// TwinCAT 3 PLC project VFD
// Title: Modbus
// Company: HuynhPhuc
// ProjectVersion: 0.0.0.0
// ProgramVersion: 3.1.4024.0
// libraries:
//   Tc2_ModbusRTU, * (Beckhoff Automation GmbH)
//   Tc2_Standard, * (Beckhoff Automation GmbH)
//   Tc2_System, * (Beckhoff Automation GmbH)
//   Tc2_Utilities, * (Beckhoff Automation GmbH)
//   Tc3_Module, * (Beckhoff Automation GmbH)
// project tree:
//   / Class Diagram.TcCD (not stored), GVL.TcGVL, Machine.TcTTO
//   DUT/Common/ U_Word2Int.TcDUT (not stored)
//   DUT/File Logger/ E_FileLoggerAddLogsState.TcDUT, E_FileLoggerInitState.TcDUT (not stored), E_FileLoggerSetNewPathState.TcDUT (not stored), E_FileLoggerState.TcDUT (not stored)
//   DUT/M_Driver/ E_VfdMdriverFaultInfor.TcDUT (not stored)
//   DUT/Universal_Modbus/ E_ModbusFunction.TcDUT, E_ModBusMasterState.TcDUT, E_ModbusMasterStateRun.TcDUT
//   DUT/VFD/ E_VFD_State.TcDUT, E_VFD_Status.TcDUT (not stored)
//   DUT/Visu/ E_VisuCtrlVfdState.TcDUT (not stored), ST_VisuCtrlVfdFrame.TcDUT (not stored)
//   FC/ FC_ScaleValue.TcPOU (not stored), FUN_MergeLongStrings10.TcPOU, FUN_MergeStrings10.TcPOU, FUN_MergeStrings3.TcPOU, FUN_MergeStrings4.TcPOU, FUN_MergeStrings5.TcPOU, FUN_MergeStrings6.TcPOU, F_InRange.TcPOU
//   POUs/EmkoTemperature/ FB_TemperatureRelativeHumiditySensor_Emko.TcPOU
//   POUs/File Logger/ FB_FileLogger.TcPOU, I_FileLogger.TcIO (not stored)
//   POUs/ Prg_Machine.TcPOU
//   POUs/Universal Modbus RTU/ FB_ModbusMaster.TcPOU, FB_ModbusSlave.TcPOU, I_ModbusSlave.TcIO
//   POUs/VFD/ FB_UniversalVFDModbus.TcPOU, FB_VFD_ABB_ACS480.TcPOU, FB_VFD_Mdriver.TcPOU, I_UniversalVFD.TcIO
//   TEST/ FB_ModbusMaster_Test.TcPOU, FB_ModbusSlave_Test.TcPOU, FB_UniversalVFDModbus_Ex.TcPOU, FB_UniversalVFDModbus_Test.TcPOU, PGR_Test.TcPOU, README.TcPOU
// real-time tasks:
//   TASK Machine: cycle T#10ms, priority 20, ADS port 350
// I/O:
//   DEVICE Device 1 (NOV-DP-RAM) (disabled)
//   DEVICE Device 4 (COM Port) (disabled)

CONFIGURATION VFD
    RESOURCE PLC ON TwinCAT3
        TASK Machine(INTERVAL := T#10ms, PRIORITY := 20);
    END_RESOURCE
END_CONFIGURATION

// ---- DUT/File Logger/E_FileLoggerAddLogsState.TcDUT
{attribute 'strict'}
TYPE E_FileLoggerAddLogsState :
(
	FILE_LOGGER_ADD_LOGS_OPEN 			:= 0,	(* Opening file *)
	FILE_LOGGER_ADD_LOGS_WRITTE			:= 10,	(* Writting log from buffer to file *)
	FILE_LOGGER_ADD_LOGS_WRITTE_DONE	:= 20,	(* Writting log from buffer to file done *)
	FILE_LOGGER_ADD_LOGS_CLOSE 			:= 30,	(* Closing file *)
	FILE_LOGGER_ADD_LOGS_CLEAR			:= 40	(* Clearing buffer *)
);
END_TYPE

// ---- DUT/Universal_Modbus/E_ModbusFunction.TcDUT
{attribute 'qualified_only'}
TYPE E_ModbusFunction :
(	
	ReadCoils	:= 1,
	ReadDisCreteInputs := 2,
	ReadHoldingRegisters := 3, 
	ReadInputRegisters := 4,
	WriteSingleCoil := 5,
	WriteSingleRegister := 6,
	WriteMultipleCoils := 15,
	WriteMultipleRegisters := 16
) WORD;
END_TYPE

// ---- DUT/Universal_Modbus/E_ModBusMasterState.TcDUT
{attribute 'qualified_only'}
{attribute 'strict'}
TYPE E_ModBusMasterState :
(
	Uninitialized := 0,//0
	Initializing := 10,//10
	Ready	:= 20	,//20
	Running		:= 30,//30
	Stop		:= 200,//200
	Stop_done	:= 210//210
	
);
END_TYPE

// ---- DUT/Universal_Modbus/E_ModbusMasterStateRun.TcDUT
{attribute 'qualified_only'}
{attribute 'strict'}
TYPE E_ModbusMasterStateRun :
(
	CheckNumberSlaveRegistered 	:=0, 
	SetParametersRead 	:= 10,
	SendRequestRead		:= 20,
	WaitReadRespond	:= 40,
	ConvertRawData	:= 50,
	ReturnReadDone		:=60,
	
	SetParametersWrite 	:= 70,
	SendRequestWrite	:= 80,
	WaitWriteRespond := 90,
	ReturnWriteDone	:=120,

	
	notKnow			:= 210

);
END_TYPE

// ---- DUT/VFD/E_VFD_State.TcDUT
{attribute 'strict'}
{attribute 'to_string'}
TYPE E_VFD_State :
(
	VFD_ABORTING := -50,
	VFD_UNINITIALIZED := 0,
	VFD_INITIALIZING	:= 10,
	VFD_READY_INITIALIZED := 20,
	VFD_IDLE		:= 30,
	VFD_RUN_FORWARD	:= 40,
	VFD_RUN_FORWARD_DONE	:= 45,
	VFD_RUN_REVERSE	:= 50,
	VFD_RUN_REVERSE_DONE := 55,
	VFD_STOP		:= 60,
	VFD_STOP_DONE	:= 70,
	VFD_RESET	:= 80,
	VFD_RESET_DONE	:= 90
)INT;
END_TYPE

// ---- GVL.TcGVL

VAR_GLOBAL
	
	fbMachineLogger 						: FB_FileLogger;
	fbMachineTime							: FB_LocalSystemTime; 			
END_VAR

// ---- POUs/Universal Modbus RTU/I_ModbusSlave.TcIO
INTERFACE I_ModbusSlave

PROPERTY AddressRead : POINTER TO WORD
GET
END_GET
END_PROPERTY

PROPERTY AddressWrite : Pointer to Word
GET
END_GET
END_PROPERTY

METHOD Convert : BOOL
VAR_INPUT
	iRegionNo	:	INT;
	pReadData	:	POINTER TO word;
END_VAR
END_METHOD

METHOD FirstCycle 
VAR_INPUT
	sName : STRING;
	iUnitID : BYTE ; // modbus address of the device : 1- 255
END_VAR
END_METHOD

PROPERTY ModbusErrorID : MODBUS_ERRORS
GET
END_GET
SET
END_SET
END_PROPERTY

PROPERTY Name : STRING
GET
END_GET
SET
END_SET
END_PROPERTY

PROPERTY NumAddRegionRead : UINT
GET
END_GET
END_PROPERTY

PROPERTY NumAddRegionWrite : Uint
GET
END_GET
END_PROPERTY

PROPERTY UnitID : BYTE
GET
END_GET
SET
END_SET
END_PROPERTY

END_INTERFACE

// ---- POUs/VFD/I_UniversalVFD.TcIO
INTERFACE I_UniversalVFD


PROPERTY Active : REFERENCE TO  bool
GET
END_GET
END_PROPERTY

PROPERTY AcVoltageToMotor : Reference to lreal
GET
END_GET
END_PROPERTY


PROPERTY Busy : reference to bool
GET
END_GET
END_PROPERTY

PROPERTY Current : reference to lreal
GET
END_GET
END_PROPERTY

PROPERTY DcVoltage : Reference to lreal
GET
END_GET
END_PROPERTY


PROPERTY Error : REFERENCE to bool
GET
END_GET
END_PROPERTY


PROPERTY ErrorID : reference to UDINT
GET
END_GET
END_PROPERTY

PROPERTY HzActual : REFERENCE TO  LReal
GET
END_GET
END_PROPERTY

PROPERTY HzControl : reference to LReal
GET
END_GET
END_PROPERTY


PROPERTY InHz : bool
GET
END_GET
END_PROPERTY

PROPERTY isRunForward : bool
GET
END_GET
END_PROPERTY


PROPERTY IsRunning : bool
GET
END_GET
END_PROPERTY

PROPERTY isRunReverse : bool
GET
END_GET
END_PROPERTY

PROPERTY isStop : bool
GET
END_GET
END_PROPERTY

METHOD MR_Abort : BOOL
VAR_INPUT
END_VAR
END_METHOD

METHOD MR_Init : bool
VAR_INPUT
END_VAR
END_METHOD

METHOD MR_Reset : BOOL
VAR_INPUT
END_VAR
END_METHOD

//must stop before call run reverse or forward
METHOD MR_RunForward : BOOL// carefully about this state , it only into run forward if estatus = VFD_STATUS_RUNNING_FORWARD or it return True
VAR_INPUT
	hz : LREAL;
END_VAR
END_METHOD

METHOD MR_RunReverse : BOOL// must stop before call run reverse or forward
VAR_INPUT
	hz : LREAL; // >0 and < 50;
END_VAR
END_METHOD

METHOD MR_Stop : BOOL
VAR_INPUT
END_VAR
END_METHOD

PROPERTY Name : STRING
GET
END_GET
SET
END_SET
END_PROPERTY


PROPERTY Overload : reference TO BOOL
GET
END_GET
END_PROPERTY


PROPERTY PowerKw : REFERENCE TO LREAL
GET
END_GET
END_PROPERTY

PROPERTY Speed : Reference to lreal
GET
END_GET
END_PROPERTY


PROPERTY State : reference to E_Vfd_State
GET
END_GET
END_PROPERTY


PROPERTY Status : reference to E_VFD_Status
GET
END_GET
END_PROPERTY

PROPERTY timeStopDelay : time
GET
END_GET
SET
END_SET
END_PROPERTY

PROPERTY Torque : reference to lreal
GET
END_GET
END_PROPERTY

PROPERTY TotalKwh : reference to lreal
GET
END_GET
END_PROPERTY

PROPERTY Warning : reference to bool
GET
END_GET
END_PROPERTY

END_INTERFACE

// ---- POUs/File Logger/FB_FileLogger.TcPOU
(* 
:Description: This function block allows to log the data to txt file
*)
FUNCTION_BLOCK FB_FileLogger IMPLEMENTS I_FileLogger
VAR CONSTANT
	iBUFFER_SIZE : UINT := 255;
END_VAR
VAR
	sName : STRING;
	
	(* First cycle bits used for selecting file logging mode *)
	bAddTimeStamp				: BOOL;
	bAddHeader					: BOOL;
	
	(* Internal status *)
	bActive 					: BOOL;						(*  *)
	bBusy						: BOOL;						(*  *)
	bError						: BOOL;						(*  *)
	iErrorID					: UDINT;					(*  *)
	
	eFileLoggerState 			: E_FileLoggerState;		(*  *)
	eFileLoggerInitState 		: E_FileLoggerInitState;	(*  *)
	eFileLoggerAddLogsState		: E_FileLoggerAddLogsState; (*  *)
	eFileLoggerSetNewPathState 	: E_FileLoggerSetNewPathState;
	
	(* Internal parameters *)
	sFileName 					: STRING;					(*  *)
	sFileDir					: STRING;					(*  *)
	sFilePath					: STRING;					(*  *)
	
	hFile						: UINT;						(*  *)
	sAmsNetId					: T_AmsNetID;				(*  *)
	stTime						: TIMESTRUCT;				(*  *)
	sTime						: STRING;					(*  *)
	sFileDate					: STRING;									(*  *)
	sLogMessage					: STRING;									(*  *)
	
	(* Buffer arrays *)
	iCurrentBufferLine			: UINT := 1;								(*  *)
	iCurrentBufferLineForFile	: UINT := 1;								(*  *)
	arrMessageBuffer 			: ARRAY [1..iBUFFER_SIZE] OF STRING(300);	(*  *)
	arrMessageBufferPresence	: ARRAY [1..iBUFFER_SIZE] OF BOOL(255);		(*  *)
	
	(* Function blocks - time handling*)
	//fbGetTime					: NT_GetTime;				(*  *)
	
	(* Function blocks - file handling *)
	fbFileOpen					: FB_FileOpen;				(*  *)
	fbFileClose					: FB_FileClose;				(*  *)
	fbCreateDir					: FB_CreateDir;				(*  *)
	fbFilePuts					: FB_FilePuts;				(*  *)
END_VAR

bActive := eFileLoggerState >= FILE_LOGGER_READY;

IF fbMachineTime.bValid THEN
	stTime := fbMachineTime.systemTime;
	sTime := SYSTEMTIME_TO_STRING(stTime);
	
END_IF

StateMachine();

PROPERTY Active : REFERENCE TO BOOL
GET
Active REF= bActive;
END_GET
END_PROPERTY

PROPERTY AmsNetId : STRING
GET
AmsNetID := sAmsNetId;
END_GET
SET
sAmsNetId := AmsNetId;
END_SET
END_PROPERTY

PROPERTY Busy : REFERENCE TO BOOL
GET
Busy REF= bBusy;
END_GET
END_PROPERTY

PROPERTY Error : REFERENCE TO BOOL
GET
Error REF= bError;
END_GET
END_PROPERTY

PROPERTY ErrorID : REFERENCE TO UDINT
GET
ErrorID REF= iErrorID;
END_GET
END_PROPERTY

PROPERTY FileDir : STRING
GET
FileDir := sFileDir;
END_GET
SET
sFileDir := FileDir;
END_SET
END_PROPERTY

PROPERTY FileName : STRING
GET
FileName := sFileName;
END_GET
SET
sFileName := FileName;
END_SET
END_PROPERTY

METHOD M_ResetParameters : BOOL
VAR_INPUT
END_VAR
fbCreateDir( bExecute := FALSE);
fbFileOpen( bExecute := FALSE);
fbFilePuts( bExecute := FALSE);
fbFileClose( bExecute := FALSE);

FOR iCurrentBufferLine := 1 TO iBUFFER_SIZE BY 1 DO
	MEMSET(ADR(arrMessageBuffer[iCurrentBufferLine]),0,SIZEOF(arrMessageBuffer[iCurrentBufferLine]));
	arrMessageBufferPresence[iCurrentBufferLine] := FALSE;
END_FOR

iCurrentBufferLine := 1;
iCurrentBufferLineForFile := 1;

bError 		:= FALSE;
iErrorID 	:= 0;

MEMSET(ADR(sLogMessage),0,SIZEOF(sLogMessage));

eFileLoggerInitState := 0;
eFileLoggerAddLogsState := 0;
END_METHOD

METHOD M_SetNewPath : BOOL
VAR_INPUT
END_VAR
CASE eFileLoggerSetNewPathState OF
	FILE_LOGGER_SET_NEW_PATH_CHANGE_PATH:
		M_SetNewPath := FALSE;
		sFilePath := CONCAT(STR1 := sFileDir, STR2 := sFileName);
		
		eFileLoggerSetNewPathState := FILE_LOGGER_SET_NEW_PATH_DONE;
	
	FILE_LOGGER_SET_NEW_PATH_DONE:
		M_SetNewPath := TRUE;
		eFileLoggerSetNewPathState := FILE_LOGGER_SET_NEW_PATH_CHANGE_PATH;
			
END_CASE
END_METHOD

METHOD MR_Abort : BOOL
IF eFileLoggerState >= FILE_LOGGER_READY THEN
	bBusy := TRUE;
	MR_Abort := FALSE;
	eFileLoggerState := FILE_LOGGER_ABORTING;
	
ELSIF eFileLoggerState = FILE_LOGGER_UNINITIALIZED THEN
	bBusy := FALSE;
	MR_Abort := TRUE;
	
END_IF
END_METHOD

METHOD MR_AddLogs : BOOL
VAR_INPUT
	sLogMessage 	: STRING;		
	
END_VAR
VAR
	sCurrentTime 	: STRING;
	sCurrentDate	: STRING;
	sLog			: STRING(300);
	
END_VAR
IF iCurrentBufferLine >= iBUFFER_SIZE THEN	
	iCurrentBufferLine := 1;
		
ELSE
	sCurrentDate := LEFT(sTime,10);
	sCurrentTime := RIGHT(sTime,12);
	MEMSET(ADR(sLog),0,SIZEOF(sLog));
	
	IF bAddTimeStamp THEN
		sLog := FUN_MergeStrings6(sCurrentDate,'$t',sCurrentTime,'$t',sLogMessage,'$n'); 
	ELSE
		sLog := CONCAT(sLogMessage,'$n'); 
	END_IF
	
	MEMSET(ADR(arrMessageBuffer[iCurrentBufferLine]),0,SIZEOF(arrMessageBuffer[iCurrentBufferLine]));
	arrMessageBuffer[iCurrentBufferLine] := sLog;
	iCurrentBufferLine := iCurrentBufferLine + 1;
	
	MR_AddLogs := TRUE;
	
END_IF
END_METHOD

METHOD MR_FirstCycle : BOOL
VAR_INPUT
	sName 			: STRING;
	sFileDir		: STRING(255);
	sFileName		: STRING(255);
	sAmsNetId		: T_AmsNetID;
	bAddTimeStamp	: BOOL;
	bAddHeader		: BOOL;
END_VAR
THIS^.sName := sName;
THIS^.sFileDir := sFileDir;
THIS^.sFileName := sFileName;
THIS^.sAmsNetId := sAmsNetId;
THIS^.bAddTimeStamp := bAddTimeStamp;
THIS^.bAddHeader := bAddHeader;

M_SetNewPath();
END_METHOD

METHOD MR_Init : BOOL
VAR_INPUT
END_VAR
IF eFileLoggerState = FILE_LOGGER_UNINITIALIZED THEN
	bBusy := TRUE;
	MR_Init := FALSE;
	eFileLoggerState := FILE_LOGGER_INITIALIZING;
	
ELSIF eFileLoggerState >= FILE_LOGGER_READY THEN
	bBusy := FALSE;
	MR_Init := TRUE;
	
END_IF
END_METHOD

METHOD MR_Reset : BOOL
IF eFileLoggerState >= FILE_LOGGER_IDLE AND eFileLoggerState <> FILE_LOGGER_METHOD_DONE THEN
	bBusy := TRUE;
	MR_Reset := FALSE;
	eFileLoggerState := FILE_LOGGER_RESET;	

ELSIF eFileLoggerState = FILE_LOGGER_METHOD_DONE THEN
	bBusy := FALSE;
	MR_Reset := TRUE;

END_IF
END_METHOD

METHOD MR_SelectPath : BOOL
VAR_INPUT
	sFileDir								: STRING; 			(* CSV source file directory name *)
	sFileName 								: STRING; 			(* CSV source file name *)
END_VAR
IF eFileLoggerState = FILE_LOGGER_IDLE THEN
	THIS^.sFileDir := sFileDir;	
	THIS^.sFileName := sFileName;	
	bBusy := TRUE;
	MR_SelectPath := FALSE;
	eFileLoggerState := FILE_LOGGER_SELECT_PATH;
	
ELSIF eFileLoggerState = FILE_LOGGER_METHOD_DONE THEN
	bBusy := FALSE;
	MR_SelectPath := TRUE;
	
END_IF
END_METHOD

METHOD PROTECTED MS_Aborting
fbCreateDir( bExecute := FALSE);
fbFileOpen( bExecute := FALSE);
fbFilePuts( bExecute := FALSE);
fbFileClose( bExecute := FALSE);
//fbGetTime( START := FALSE);

FOR iCurrentBufferLine := 1 TO iBUFFER_SIZE BY 1 DO
	MEMSET(ADR(arrMessageBuffer[iCurrentBufferLine]),0,SIZEOF(arrMessageBuffer[iCurrentBufferLine]));
	arrMessageBufferPresence[iCurrentBufferLine] := FALSE;
	
END_FOR

iCurrentBufferLine := 1;
iCurrentBufferLineForFile := 1;

MEMSET(ADR(sTime),0,SIZEOF(sTime));
MEMSET(ADR(sFileDate),0,SIZEOF(sFileDate));
MEMSET(ADR(sLogMessage),0,SIZEOF(sLogMessage));

stTime.wDay 			:= 0;
stTime.wDayOfWeek 		:= 0;
stTime.wHour 			:= 0;
stTime.wMilliseconds 	:= 0;
stTime.wMinute 			:= 0;
stTime.wMonth 			:= 0;
stTime.wSecond 			:= 0;
stTime.wYear 			:= 0;

bActive		:= FALSE;
bBusy 		:= FALSE;
bError 		:= FALSE;
iErrorID 	:= 0;

eFileLoggerInitState := FILE_LOGGER_INIT_GET_TIME;
eFileLoggerAddLogsState := FILE_LOGGER_ADD_LOGS_OPEN;
eFileLoggerState := FILE_LOGGER_UNINITIALIZED;
END_METHOD

METHOD PROTECTED MS_AddLogs
CASE eFileLoggerAddLogsState OF
	FILE_LOGGER_ADD_LOGS_OPEN:
		IF NOT fbFileOpen.bError THEN
			fbFileOpen( sNetId 		:= sAmsNetId,
						sPathName 	:= FUN_MergeStrings4(sStr1 := sFilePath,'_',LEFT(sTime,10),'.txt'),
						bExecute 	:= TRUE,
						tTimeout	:= DEFAULT_ADS_TIMEOUT,
						nMode		:= FOPEN_MODEAPPEND OR FOPEN_MODEPLUS);
							
			IF NOT fbFileOpen.bBusy THEN
				fbFileOpen(bExecute := FALSE);				
				hFile := fbFileOpen.hFile;;
				eFileLoggerAddLogsState := FILE_LOGGER_ADD_LOGS_WRITTE;
			
			END_IF
		ELSE
			fbFileOpen( bExecute := FALSE);
			bError := fbFileOpen.bError;
			iErrorID := fbFileOpen.nErrId;

		END_IF
	

	FILE_LOGGER_ADD_LOGS_WRITTE:
		IF NOT fbFilePuts.bError THEN
			fbFilePuts( sNetId		:= sAmsNetId,
						hFile 		:= hFile,
						sLine 		:= arrMessageBuffer[iCurrentBufferLineForFile],
						bExecute 	:= TRUE,
						tTimeout 	:= DEFAULT_ADS_TIMEOUT);	
					
			IF NOT fbFilePuts.bBusy THEN				
				eFileLoggerAddLogsState := FILE_LOGGER_ADD_LOGS_WRITTE_DONE;
				
			END_IF
			
		ELSE
			fbFilePuts( bExecute := FALSE);
			bError := fbFilePuts.bError;
			iErrorID := fbFilePuts.nErrId;
			
		END_IF	

		
	FILE_LOGGER_ADD_LOGS_WRITTE_DONE:
		fbFilePuts( bExecute := FALSE);	
		iCurrentBufferLineForFile := iCurrentBufferLineForFile + 1;	
		
		IF iCurrentBufferLineForFile >= iBUFFER_SIZE THEN
			iCurrentBufferLineForFile := 1;
		ELSIF iCurrentBufferLineForFile < iCurrentBufferLine THEN
			eFileLoggerAddLogsState := FILE_LOGGER_ADD_LOGS_WRITTE;
		ELSIF iCurrentBufferLineForFile >= iCurrentBufferLine THEN
			eFileLoggerAddLogsState := FILE_LOGGER_ADD_LOGS_CLOSE;
		END_IF;

	
	FILE_LOGGER_ADD_LOGS_CLOSE:
		IF NOT fbFileClose.bError THEN
			fbFileClose(	sNetId := sAmsNetId,
							hFile := hFile,
							bExecute := TRUE,
							tTimeout := DEFAULT_ADS_TIMEOUT);
							
			IF NOT fbFileClose.bBusy THEN
				fbFileClose( bExecute := FALSE);
				eFileLoggerAddLogsState := FILE_LOGGER_ADD_LOGS_OPEN;
				eFileLoggerState := FILE_LOGGER_IDLE;

			END_IF
		ELSE
			bError := fbFileClose.bError;
			iErrorID := fbFileClose.nErrId;
			fbFileClose( bExecute := FALSE);
			
		END_IF
		
END_CASE
END_METHOD

METHOD PROTECTED MS_Idle
VAR_INPUT
END_VAR
IF iCurrentBufferLineForFile < iCurrentBufferLine THEN
	eFileLoggerState := FILE_LOGGER_ADD_LOGS;

END_IF
END_METHOD

METHOD PROTECTED MS_Initializing //C:\TwinCAT\log\filelog.txt
CASE eFileLoggerInitState OF
	FILE_LOGGER_INIT_CREATE_DIR:
		fbCreateDir(sNetId 		:= sAmsNetId,
					sPathName 	:= sFileDir,
					bExecute 	:= TRUE,
					tTimeout 	:= DEFAULT_ADS_TIMEOUT);
					
		IF NOT fbCreateDir.bBusy THEN
			eFileLoggerInitState := FILE_LOGGER_INIT_GET_TIME;
			fbCreateDir( bExecute := FALSE);
			
		END_IF
		
	FILE_LOGGER_INIT_GET_TIME:
		IF fbMachineTime.bValid THEN
			stTime := fbMachineTime.systemTime;
			sTime := SYSTEMTIME_TO_STRING(stTime);
			sFileDate := LEFT(sTime,10);
			eFileLoggerInitState := FILE_LOGGER_INIT_CREATE_FILE;
			
		END_IF
		
	FILE_LOGGER_INIT_CREATE_FILE:
		IF NOT fbFileOpen.bError THEN
			fbFileOpen( sNetId 		:= sAmsNetId,
						sPathName 	:= FUN_MergeStrings4(sFilePath,'_',LEFT(sTime,10),'.txt'),
						bExecute 	:= TRUE,
						tTimeout	:= DEFAULT_ADS_TIMEOUT,
						nMode		:= FOPEN_MODEAPPEND OR FOPEN_MODEPLUS);
							
			IF NOT fbFileOpen.bBusy THEN
				hFile := fbFileOpen.hFile;
				fbFileOpen(bExecute := FALSE);		
				
				IF bAddHeader THEN 
					eFileLoggerInitState := FILE_LOGGER_INIT_ADD_HEADER;
					
				ELSE
					eFileLoggerInitState := FILE_LOGGER_INIT_CLOSE_FILE;
					
				END_IF							
			END_IF
		ELSE
			bError := fbFileOpen.bError;
			iErrorID := fbFileOpen.nErrId;
			fbFileOpen( bExecute := FALSE);
			
		END_IF
		
	FILE_LOGGER_INIT_ADD_HEADER:
	
		IF NOT fbFilePuts.bError THEN
			fbFilePuts(	sNetId := sAmsNetId,
						hFile := hFile,
						sLine := CONCAT('----- Logger file initialized at ',CONCAT(LEFT(sTime,23),' ----- $n')),
						bExecute := TRUE,
						tTimeout := DEFAULT_ADS_TIMEOUT);

			IF NOT fbFilePuts.bBusy THEN
				eFileLoggerInitState := FILE_LOGGER_INIT_CLOSE_FILE;
				fbFilePuts( bExecute := FALSE);
				
			END_IF	
		ELSE
			bError := fbFilePuts.bError;
			iErrorID := fbFilePuts.nErrId;
			fbFilePuts( bExecute := FALSE);
			
		END_IF
	
	FILE_LOGGER_INIT_CLOSE_FILE:
		IF NOT fbFileClose.bError THEN
			fbFileClose( sNetId 		:= sAmsNetId,
							hFile 		:= hFile,
							bExecute 	:= TRUE,
							tTimeout 	:= DEFAULT_ADS_TIMEOUT);
							
			IF NOT fbFileClose.bBusy THEN
				eFileLoggerInitState := FILE_LOGGER_INIT_DONE;
				fbFileClose( bExecute := FALSE);
				
			END_IF
		ELSE
			bError := fbFileClose.bError;
			iErrorID := fbFileClose.nErrId;
			fbFileClose( bExecute := FALSE);
			
		END_IF
	
	FILE_LOGGER_INIT_DONE:
		eFileLoggerInitState := FILE_LOGGER_INIT_CREATE_DIR;
		eFileLoggerState := FILE_LOGGER_IDLE;
		
END_CASE
END_METHOD

METHOD PROTECTED MS_MethodDone
VAR_INPUT
END_VAR
IF NOT bBusy THEN
	eFileLoggerState := FILE_LOGGER_IDLE;

END_IF
END_METHOD

METHOD PROTECTED MS_Ready
VAR_INPUT
END_VAR
eFileLoggerState := FILE_LOGGER_IDLE;
END_METHOD

METHOD PROTECTED MS_Reset
VAR_INPUT
END_VAR
IF M_ResetParameters() THEN
	eFileLoggerState := FILE_LOGGER_METHOD_DONE;
	
END_IF
END_METHOD

METHOD MS_SelectPath : BOOL
VAR_INPUT
END_VAR
IF M_SetNewPath() THEN
	eFileLoggerState := FILE_LOGGER_METHOD_DONE;
	
END_IF
END_METHOD

METHOD PROTECTED MS_Uninitialized
;
END_METHOD

PROPERTY Name : STRING
GET
Name := sName;
END_GET
SET
sName := Name;
END_SET
END_PROPERTY

METHOD PROTECTED StateMachine
CASE eFileLoggerState OF
	FILE_LOGGER_UNINITIALIZED:
		MS_Uninitialized();
		
	FILE_LOGGER_INITIALIZING:
		MS_Initializing();
		
	FILE_LOGGER_IDLE:
		MS_Idle();
		
	FILE_LOGGER_ADD_LOGS:
		MS_AddLogs();	
		
	FILE_LOGGER_RESET:
		MS_Reset();
		
	FILE_LOGGER_METHOD_DONE:
		MS_MethodDone();
	
	FILE_LOGGER_ABORTING:
		MS_Aborting();
	
END_CASE
END_METHOD

END_FUNCTION_BLOCK

// ---- FC/FUN_MergeStrings6.TcPOU
(* 
:Description: This function is used to merge 6 strings
*)
FUNCTION FUN_MergeStrings6 : STRING(300)
VAR_INPUT
	sStr1	: STRING;		(* First string in merge row *)
	sStr2	: STRING;		(* Second string in merge row *)
	sStr3	: STRING;		(* Third string in merge row *)
	sStr4	: STRING;		(* Fourth string in merge row *)
	sStr5	: STRING;		(* Fifth string in merge row *)
	sStr6	: STRING;		(* Sixth string in merge row *)
END_VAR
(*
Version history:

+-------------+------------+----------------+----------+------------------------------------------+
|Date         | Version    | created under  | Author   | Remark                                   |
+=============+============+================+==========+==========================================+
|2022-06      | 1.0.0.0    | V3.1.4024.22   | ADS      | Function created    		              |
+-------------+------------+----------------+----------+------------------------------------------+

*)

FUN_MergeStrings6 := CONCAT(sStr1,sStr2);
FUN_MergeStrings6 := CONCAT(FUN_MergeStrings6, sStr3);
FUN_MergeStrings6 := CONCAT(FUN_MergeStrings6, sStr4);
FUN_MergeStrings6 := CONCAT(FUN_MergeStrings6, sStr5);
FUN_MergeStrings6 := CONCAT(FUN_MergeStrings6, sStr6);

END_FUNCTION

// ---- FC/FUN_MergeStrings4.TcPOU
(* 
:Description: This function is used to merge 5 strings
*)
FUNCTION FUN_MergeStrings4 : STRING
VAR_INPUT
	sStr1	: STRING;			(* Fifth string in merge row *)
	sStr2	: STRING;			(* Fourth string in merge row *)
	sStr3	: STRING;			(* Fourth string in merge row *)
	sStr4	: STRING;			(* Fourth string in merge row *)

END_VAR

FUN_MergeStrings4 := CONCAT(sStr1,sStr2);
FUN_MergeStrings4 := CONCAT(FUN_MergeStrings4,sStr3);
FUN_MergeStrings4 := CONCAT(FUN_MergeStrings4,sStr4);

END_FUNCTION

// ---- FC/FUN_MergeLongStrings10.TcPOU
(* 
:Description: This function is used to merge 10 long strings
*)
FUNCTION FUN_MergeLongStrings10 : STRING(2000)
VAR_INPUT
	sStr1	: STRING(2000);
	sStr2	: STRING(2000);
	sStr3	: STRING(2000);
	sStr4	: STRING(2000);
	sStr5	: STRING(2000);
	sStr6	: STRING(2000);
	sStr7	: STRING(2000);
	sStr8	: STRING(2000);
	sStr9	: STRING(2000);
	sStr10	: STRING(2000);
END_VAR
VAR
	sStrTemp1 :	STRING(2000);
	sStrTemp2 :	STRING(2000);
END_VAR
(*
Version history:

+-------------+------------+----------------+----------+------------------------------------------+
|Date         | Version    | created under  | Author   | Remark                                   |
+=============+============+================+==========+==========================================+
|2021-11      | 1.0.0.0    | V3.1.4024.22   | ADBO     | Function created		                  |
+-------------+------------+----------------+----------+------------------------------------------+

*)

CONCAT2(ADR(sStr1),ADR(sStr2),ADR(sStrTemp1),SIZEOF(sStrTemp1));
CONCAT2(ADR(sStrTemp1),ADR(sStr3),ADR(sStrTemp2),SIZEOF(sStrTemp2));
CONCAT2(ADR(sStrTemp2),ADR(sStr4),ADR(sStrTemp1),SIZEOF(sStrTemp1));
CONCAT2(ADR(sStrTemp1),ADR(sStr5),ADR(sStrTemp2),SIZEOF(sStrTemp2));
CONCAT2(ADR(sStrTemp2),ADR(sStr6),ADR(sStrTemp1),SIZEOF(sStrTemp1));
CONCAT2(ADR(sStrTemp1),ADR(sStr7),ADR(sStrTemp2),SIZEOF(sStrTemp2));
CONCAT2(ADR(sStrTemp2),ADR(sStr8),ADR(sStrTemp1),SIZEOF(sStrTemp1));
CONCAT2(ADR(sStrTemp1),ADR(sStr9),ADR(sStrTemp2),SIZEOF(sStrTemp2));
CONCAT2(ADR(sStrTemp2),ADR(sStr10),ADR(FUN_MergeLongStrings10),SIZEOF(FUN_MergeLongStrings10));

END_FUNCTION

// ---- FC/FUN_MergeStrings10.TcPOU
(* 
:Description: This function is used to merge 10 strings
*)
FUNCTION FUN_MergeStrings10 : STRING
VAR_INPUT
	sStr1	: STRING;		(* First string in merge row *)
	sStr2	: STRING;		(* Second string in merge row *)
	sStr3	: STRING;		(* Third string in merge row *)
	sStr4	: STRING(500);	(* Fourth string in merge row *)
	sStr5	: STRING(500);	(* Fifth string in merge row *)
	sStr6	: STRING(500);	(* Sixth string in merge row *)
	sStr7	: STRING(500);	(* Seventh string in merge row *)
	sStr8	: STRING;		(* Eight string in merge row *)
	sStr9	: STRING;		(* Ninth string in merge row *)
	sStr10	: STRING;		(* Tenth string in merge row *)
END_VAR
(*
Version history:

+-------------+------------+----------------+----------+------------------------------------------+
|Date         | Version    | created under  | Author   | Remark                                   |
+=============+============+================+==========+==========================================+
|2021-11      | 1.0.0.0    | V3.1.4024.22   | ADBO     | Function created      		              |
+-------------+------------+----------------+----------+------------------------------------------+

*)

FUN_MergeStrings10 := CONCAT(sStr1,sStr2);
FUN_MergeStrings10 := CONCAT(FUN_MergeStrings10,sStr3);
FUN_MergeStrings10 := CONCAT(FUN_MergeStrings10,sStr4);
FUN_MergeStrings10 := CONCAT(FUN_MergeStrings10,sStr5);
FUN_MergeStrings10 := CONCAT(FUN_MergeStrings10,sStr6);
FUN_MergeStrings10 := CONCAT(FUN_MergeStrings10,sStr7);
FUN_MergeStrings10 := CONCAT(FUN_MergeStrings10,sStr8);
FUN_MergeStrings10 := CONCAT(FUN_MergeStrings10,sStr9);
FUN_MergeStrings10 := CONCAT(FUN_MergeStrings10,sStr10);

END_FUNCTION

// ---- FC/FUN_MergeStrings3.TcPOU
(* 
:Description: This function is used to merge 5 strings
*)
FUNCTION FUN_MergeStrings3 : STRING
VAR_INPUT
	sStr1	: STRING;			(* Fifth string in merge row *)
	sStr2	: STRING;			(* Fourth string in merge row *)
	sStr3	: STRING;			(* Fourth string in merge row *)

END_VAR
(*
Version history:

+-------------+------------+----------------+----------+------------------------------------------+
|Date         | Version    | created under  | Author   | Remark                                   |
+=============+============+================+==========+==========================================+
|2022-06      | 1.0.0.0    | V3.1.4024.22   | ADS      | Function created    		              |
+-------------+------------+----------------+----------+------------------------------------------+

*)

FUN_MergeStrings3 := CONCAT(sStr1,sStr2);
FUN_MergeStrings3 := CONCAT(FUN_MergeStrings3,sStr3);

END_FUNCTION

// ---- FC/FUN_MergeStrings5.TcPOU
(* 
:Description: This function is used to merge 5 strings
*)
FUNCTION FUN_MergeStrings5 : STRING
VAR_INPUT
	sStr1	: STRING;		(* First string in merge row *)
	sStr2	: STRING;		(* Second string in merge row *)
	sStr3	: STRING;		(* Third string in merge row *)
	sStr4	: STRING;		(* Fourth string in merge row *)
	sStr5	: STRING;		(* Fifth string in merge row *)

END_VAR
(*
Version history:

+-------------+------------+----------------+----------+------------------------------------------+
|Date         | Version    | created under  | Author   | Remark                                   |
+=============+============+================+==========+==========================================+
|2021-11      | 1.0.0.0    | V3.1.4024.22   | ADBO     | Function created    		              |
+-------------+------------+----------------+----------+------------------------------------------+

*)

FUN_MergeStrings5 := CONCAT(sStr1,sStr2);
FUN_MergeStrings5 := CONCAT(FUN_MergeStrings5, sStr3);
FUN_MergeStrings5 := CONCAT(FUN_MergeStrings5, sStr4);
FUN_MergeStrings5 := CONCAT(FUN_MergeStrings5, sStr5);

END_FUNCTION

// ---- FC/F_InRange.TcPOU
FUNCTION F_InRange : BOOL // return true if value in [bound1, bound2] or in [bound2, bound1] else return false
VAR_INPUT
	bound1 : LREAL;
	bound2 : LREAL;
	value	: LREAL;
END_VAR
VAR
END_VAR

F_InRange := MIN(bound1, bound2)  <= value AND value <= MAX( bound1, bound2);

END_FUNCTION

// ---- POUs/EmkoTemperature/FB_TemperatureRelativeHumiditySensor_Emko.TcPOU
(*Odd or none parity bit only in model  PMDLx-x-0/0.1.1.x.x*)
FUNCTION_BLOCK FB_TemperatureRelativeHumiditySensor_Emko EXTENDS FB_ModbusSlave

VAR
	lrTemperature	: LREAL;
	lrRelativeHumidity : LREAL;
END_VAR

METHOD Convert : BOOL
VAR_INPUT
	iRegionNo	:	INT;
	pReadData	:	POINTER TO word;
END_VAR
CASE iRegionNo OF
	0:
		lrTemperature := WORD_TO_LREAL( pReadData[0])*0.01;
		lrRelativeHumidity := WORD_TO_LREAL( pReadData[1])*0.1;
END_CASE
END_METHOD

METHOD FirstCycle // must be call once time 
VAR_INPUT
	sName : STRING;
	iUnitID : BYTE ; // modbus address of the device : 1- 255
END_VAR
SUPER^.FirstCycle( sName := sName,
					iUnitID := iUnitID);
arrAddressRead[0][0] := 0;
arrAddressRead[0][1] := 2;
arrAddressRead[0][2] := E_ModbusFunction.ReadInputRegisters;
iNumAddRegionRead:= 1;
iNumAddRegionWrite := 0;
END_METHOD

PROPERTY RelativeHumidity : lreal
GET
RelativeHumidity := lrRelativeHumidity;
END_GET
END_PROPERTY

PROPERTY Temperature : lreal
GET
Temperature := lrTemperature;
END_GET
END_PROPERTY

END_FUNCTION_BLOCK

// ---- POUs/Universal Modbus RTU/FB_ModbusSlave.TcPOU
FUNCTION_BLOCK FB_ModbusSlave IMPLEMENTS I_ModbusSlave
VAR
	iUnitID	:	BYTE; // address of the Slave
	arrAddressRead	:	ARRAY [0..50] OF ARRAY [0..2] OF WORD;
	(*arrAddressRead[x][y]: +x : index of Region Read.  arrAddressRead[0]: the first region Read.
							+y:
								case y of
									0: Register address for Read
									1: Number of register for read
									2: Function Read
					 *)
	iNumAddRegionRead	:	UINT;
	
	arrAddressWrite		: ARRAY [0..20] OF ARRAY [0..10] OF WORD;// write Multiple or single register
	(* the 20 is max number of region write,
		arrAddressWrite[x][y] : +x: index of Region Read.  arrAddressRead[0]: the first region Read. 
								+y:
									case y of
										0 :  Register address for Write
										1 : number of register will be write => modbus master automatic choose Function Write( single Register or Multi Regiseter)
										2..9 : max 8 value for write
										10: Write Function : e.g E_ModbusFunction.WriteSingleCoil
															
	*)
	iNumAddRegionWrite	: UINT;
	
	bSwap			:		BOOL; // swap word receive from modbus master for convert
	sName			:		STRING;
	bFirstCycle 	: 		BOOL := TRUE;
	iModbusErrorID	:		MODBUS_ERRORS;
END_VAR

PROPERTY AddressRead : POINTER TO WORD
GET
AddressRead := ADR(arrAddressRead);
END_GET
END_PROPERTY

PROPERTY AddressWrite : POINTER TO WORD
GET
AddressWrite := ADR( arrAddressWrite);
END_GET
END_PROPERTY

METHOD Convert : BOOL
VAR_INPUT
	iRegionNo	:	INT;
	pReadData	:	POINTER TO word;
END_VAR
END_METHOD

METHOD FirstCycle // must be call once time 
VAR_INPUT
	sName : STRING;
	iUnitID : BYTE ; // modbus address of the device : 1- 255
END_VAR
THIS^.sName := sName;
THIS^.iUnitID := iUnitID;
END_METHOD

{attribute 'monitoring' := 'variable'}
PROPERTY ModbusErrorID : MODBUS_ERRORS
GET
ModbusErrorID := iModbusErrorID;
END_GET
SET
iModbusErrorID := ModbusErrorID;
END_SET
END_PROPERTY

PROPERTY Name : STRING
GET
Name := sName;
END_GET
SET
sName := Name;
END_SET
END_PROPERTY

PROPERTY NumAddRegionRead : UINT
GET
NumAddRegionRead := iNumAddRegionRead;
END_GET
END_PROPERTY

PROPERTY NumAddRegionWrite : UINT
GET
NumAddRegionWrite := iNumAddRegionWrite;
END_GET
END_PROPERTY

PROPERTY UnitID : BYTE
GET
UnitID := iUnitID;
END_GET
SET
iUnitID := UnitID;
END_SET
END_PROPERTY

END_FUNCTION_BLOCK

// ---- POUs/Prg_Machine.TcPOU
PROGRAM Prg_Machine
VAR
	fbModbusMaster	: FB_ModbusMaster;
	ABBAcs480 : FB_VFD_ABB_ACS480;
	Mdriver : fB_VFD_Mdriver;
	arrIfVFD : ARRAY[0..numberOfVFD-1] OF I_UniversalVFD;
	emkoSs	: FB_TemperatureRelativeHumiditySensor_Emko;
	bInit	: BOOL;
	bAbort : BOOL;
	bFirstCycle	: BOOL := TRUE;
	bModbusRun	: BOOL;
	hzControl	: LREAL;
	arrVfdState	: ARRAY [0..iVFDS_PER_PAGE-1] OF E_VisuCtrlVfdState; 
	arrVfdFrame	: ARRAY [0..iVFDS_PER_PAGE-1] OF ST_VisuCtrlVfdFrame;
	iloop		: UINT;
	lrTemp	: LREAL;
	lrhumidity	: LREAL;
END_VAR
VAR CONSTANT
	iVFDS_PER_PAGE : UINT := 2;
	numberOfVFD	: UINT := 2;
END_VAR

IF bFirstCycle THEN
	Mdriver.FirstCycle( sName := 'M_driver',
						iUnitID := 4 );
	ABBAcs480.FirstCycle( sName := 'ABB acs480',
							iUnitID := 5);			
	emkoSs.FirstCycle( sName := 'ss 01',
						iUnitID := 10);
	arrIfVFD[0] := Mdriver;
	arrIfVFD[1] := ABBAcs480;				
	IF fbModbusMaster.Init() THEN
		fbModbusMaster.RegisterSlave( ModbusSlave := ABBAcs480);
		fbModbusMaster.RegisterSlave( ModbusSlave := Mdriver);
		fbModbusMaster.RegisterSlave( ModbusSlave := emkoSs);
		fbModbusMaster.Timeout := 1000;
		bFirstCycle := FALSE;
	END_IF
END_IF
fbModbusMaster.Run();
fbModbusMaster();
Mdriver();
ABBAcs480();
lrTemp := emkoSs.Temperature;
lrhumidity := emkoSs.RelativeHumidity;
(*visu*)
FOR iloop := 0 TO numberOfVFD-1 DO
	arrVfdFrame[iLoop].lrCurrent		:= arrIfVFD[iloop].Current;
	arrVfdFrame[iLoop].bError			:= arrIfVFD[iloop].error;
	arrVfdFrame[iLoop].lrHz_actual		:= arrIfVFD[iloop].HzActual;
	arrVfdFrame[iLoop].eStatus			:= arrIfVFD[iloop].Status;
	arrVfdFrame[iLoop].sStatus			:= TO_STRING(arrVfdFrame[iLoop].eStatus);
	arrVfdFrame[iLoop].eState			:= arrIfVFD[iloop].State;
	arrVfdFrame[iloop].sState			:= TO_STRING(arrVfdFrame[iLoop].eState);
	arrVfdFrame[iloop].errorID			:= arrIfVFD[iloop].errorID;	
	arrVfdFrame[iloop].sName			:= arrIfVFD[iloop].Name;	
	IF arrVfdFrame[iLoop].btnReset THEN
		arrVfdFrame[iLoop].btnReset := FALSE;
		arrVfdState[iLoop] := VISU_CTRL_VFDS_RESET;
	END_IF
	
	IF arrVfdFrame[iLoop].btnAbort THEN
		arrVfdFrame[iLoop].btnAbort	:= FALSE;
		arrVfdState[iLoop] := VISU_CTRL_VFDS_ABORT;						
	END_IF	
	CASE arrVfdState[iLoop] OF
		
		VISU_CTRL_VFDS_WAIT_FOR_CMD:
			IF arrVfdFrame[iLoop].btnInit THEN
				arrVfdFrame[iLoop].btnInit	:= FALSE;
				arrVfdState[iLoop] := VISU_CTRL_VFDS_INIT;
				
			ELSIF arrVfdFrame[iLoop].btnStop THEN
				arrVfdFrame[iLoop].btnStop	:= FALSE;
				arrVfdState[iLoop] := VISU_CTRL_VFDS_STOP;
				
			ELSIF arrVfdFrame[iLoop].btnRunForward THEN
				arrVfdFrame[iLoop].btnRunForward	:= FALSE;
				arrVfdState[iLoop] := VISU_CTRL_VFDS_RUN_FORWARD;
				
			ELSIF arrVfdFrame[iLoop].btnRunReverse THEN
				arrVfdFrame[iLoop].btnRunReverse	:= FALSE;
				arrVfdState[iLoop] := VISU_CTRL_VFDS_RUN_REVERSE;						
				
			END_IF
			
		VISU_CTRL_VFDS_INIT:					
			arrIfVFD[iloop].MR_Init();
			IF arrIfVFD[iloop].Active AND NOT arrIfVFD[iloop].Busy THEN
				arrVfdState[iLoop] := VISU_CTRL_VFDS_WAIT_FOR_CMD;
			END_IF
			
		VISU_CTRL_VFDS_RESET:		 			
			arrIfVFD[iloop].MR_Reset();
			IF NOT arrIfVFD[iloop].Error AND NOT arrIfVFD[iloop].Busy THEN
				arrVfdState[iLoop] := VISU_CTRL_VFDS_WAIT_FOR_CMD;
			END_IF
		
		VISU_CTRL_VFDS_RUN_FORWARD:	
			arrIfVFD[iloop].MR_RunForward(arrVfdFrame[iLoop].lrHz_Control);		
			IF arrIfVFD[iloop].isRunForward AND NOT arrIfVFD[iloop].Busy THEN
				arrVfdState[iLoop] := VISU_CTRL_VFDS_WAIT_FOR_CMD;
			END_IF
		
		VISU_CTRL_VFDS_RUN_REVERSE:
			arrIfVFD[iloop].MR_RunReverse(arrVfdFrame[iLoop].lrHz_Control);
			IF arrIfVFD[iloop].isRunReverse AND NOT arrIfVFD[iloop].Busy THEN
				arrVfdState[iLoop] := VISU_CTRL_VFDS_WAIT_FOR_CMD;
			END_IF
			
		VISU_CTRL_VFDS_STOP:
			arrIfVFD[iloop].MR_Stop();
			IF arrIfVFD[iloop].isStop AND NOT arrIfVFD[iloop].Busy THEN
				arrVfdState[iLoop] := VISU_CTRL_VFDS_WAIT_FOR_CMD;
			END_IF
			
		VISU_CTRL_VFDS_ABORT:
			arrIfVFD[iloop].MR_Abort();
			IF NOT arrIfVFD[iloop].Active AND NOT arrIfVFD[iloop].Busy	THEN
				arrVfdState[iLoop] := VISU_CTRL_VFDS_WAIT_FOR_CMD;
			END_IF
					
	END_CASE
END_FOR

END_PROGRAM

// ---- POUs/Universal Modbus RTU/FB_ModbusMaster.TcPOU
FUNCTION_BLOCK FB_ModbusMaster //IMPLEMENTS I_UniversalUnit
VAR
	sName			:		STRING;
	bInitialized	:		BOOL;
	iScantime		:		UINT;
	iTimeout		:		UINT := 1000;//1000ms
	iErrorID		:		MODBUS_ERRORS;
	bBusy			: 		BOOL;
	bError			:		BOOL;
	iStepGeneral	: 		E_ModBusMasterState;
	iStepRunning	:		E_ModbusMasterStateRun;
	bFirstCycle		:		BOOL;
	bRun			:		BOOL;
	bStop			: 		BOOL;

	fbModbusMaster	: 		ModbusRtuMaster_PcCOM;
	//fbModbusMaster : 		ModbusRtuMasterV2_KL6x22B;
	ipModbusSlave	:		ARRAY [1..247] OF I_ModbusSlave;
	iAmountSlave	: 		UINT;
	
	iLoopSlave		:		UINT	:= 1;
	iLoopAdr		:		UINT;
	iQuantity 		: 		POINTER TO WORD;
	iMBAddr 		: 		POINTER TO WORD;
    arrData			: 		ARRAY [0..255] OF WORD;
	
	UnitId	: BYTE;
	Quantity	: WORD;
	MBAddr	: WORD;
	cbLength : UINT;
	pMemoryAddr	: POINTER TO BYTE;
	pDataWrite	: POINTER TO WORD;

	bexecute	: BOOL;
	
	tCalculateTimeRW	: TON;
	nNumberFaultRW	: UINT;
	eModbusFunction: E_ModbusFunction;
	peModbusFunction : POINTER TO WORD;
END_VAR

StateMachine();
bRun :=  iStepGeneral = E_ModBusMasterState.Running ;
bStop := iStepGeneral = E_ModBusMasterState.stop_done;
bInitialized := iStepGeneral >= E_ModBusMasterState.Ready;
iErrorID := fbModbusMaster.ErrorId;
tCalculateTimeRW(PT	:= T#10S); // for test how much time read write total

METHOD Abort : BOOL
bError := FALSE;
iErrorID := 0;
bError := FALSE;
iStepGeneral	:= E_ModBusMasterState.Uninitialized;
iStepRunning	:= E_ModbusMasterStateRun.CheckNumberSlaveRegistered;

iLoopSlave		:= 1;
iLoopAdr		:= 0;

fbModbusMaster(Execute := FALSE);

Abort := TRUE;
END_METHOD

PROPERTY AnyError : BOOL
GET
AnyError 	:= bError;
END_GET
END_PROPERTY

PROPERTY Busy : BOOL
GET
Busy := bBusy;
END_GET
END_PROPERTY

PROPERTY ErrorID : MODBUS_ERRORS
GET
ErrorID := iErrorID;
END_GET
END_PROPERTY

METHOD Init : BOOL
IF iStepGeneral = E_ModBusMasterState.Uninitialized THEN
	iStepGeneral := E_ModBusMasterState.Initializing;
END_IF

//Method output
	Init := (iStepGeneral >= E_ModBusMasterState.Ready);
END_METHOD

PROPERTY Initialized : BOOL
GET
Initialized := bInitialized;
END_GET
END_PROPERTY

PROPERTY Name : STRING
GET
Name := sName;
END_GET
SET
sName := Name;
END_SET
END_PROPERTY

PROPERTY ReadData : ARRAY [0..255] OF Word
GET
ReadData := arrData;
END_GET
END_PROPERTY

PROPERTY ReadDataSize : uint
GET
ReadDataSize := INT_TO_UINT(SIZEOF(arrData));
END_GET
END_PROPERTY

METHOD RegisterSlave : BOOL
VAR_INPUT
	ModbusSlave		:		I_ModbusSlave;
END_VAR
VAR
	iLoop	:	UINT;
	bExists	:	BOOL;
END_VAR
FOR iLoop := 1 TO iAmountSlave DO
	IF ipModbusSlave[iLoop] = ModbusSlave THEN
		bExists := TRUE;
		iLoop := iAmountSlave;// end loop for command
	END_IF
END_FOR 
IF NOT bExists THEN
	iAmountSlave := iAmountSlave + 1;
	ipModbusSlave[iAmountSlave] := ModbusSlave;
END_IF
END_METHOD

METHOD Reset : BOOL
bError := FALSE;
iErrorID := 0;
bError := FALSE;
iStepGeneral	:= E_ModBusMasterState.Uninitialized;
iStepRunning	:= E_ModbusMasterStateRun.CheckNumberSlaveRegistered;

iLoopSlave		:= 1;
iLoopAdr		:= 0;

fbModbusMaster.Execute := FALSE;

Reset := TRUE;
END_METHOD

METHOD Run : BOOL /// call from FB_modbus
IF (iStepGeneral = E_ModBusMasterState.Ready) THEN
	iStepGeneral := E_ModBusMasterState.Running;
END_IF

bRun := TRUE;
Run := (iStepGeneral >= E_ModBusMasterState.Running) AND (iStepGeneral < E_ModBusMasterState.stop);
END_METHOD

PROPERTY ScanTime : UINT
GET
ScanTime := iScantime;
END_GET
SET
iScantime := ScanTime;
END_SET
END_PROPERTY

METHOD protected StateInit : BOOL (*Unit is performing initialization*)
IF NOT bError THEN
	iStepGeneral := E_ModBusMasterState.Ready;
END_IF
END_METHOD

METHOD protected StateMachine : BOOL (*State machine of unit*)
CASE iStepGeneral OF
		E_ModBusMasterState.Uninitialized:  
			StateUninitialized();
	
		E_ModBusMasterState.Initializing: 
			StateInit();
	
		E_ModBusMasterState.Ready: 
			StateReady();
		
		E_ModBusMasterState.Running: 
			StateRunning();
						
		E_ModBusMasterState.stop:
			StateStopping();
			
		E_ModBusMasterState.stop_done:
			StateStoppingDone();
END_CASE
END_METHOD

METHOD protected StateReady : BOOL (* Unit is initialized*)
END_METHOD

METHOD PROTECTED StateRunning : BOOL (* Unit is uninitialized*)
VAR 
	

	
END_VAR
CASE iStepRunning OF
	E_ModbusMasterStateRun.CheckNumberSlaveRegistered: // Trigger
		IF iAmountSlave > 0 THEN
			iStepRunning := E_ModbusMasterStateRun.SetParametersRead;
		END_IF
					
	E_ModbusMasterStateRun.SetParametersRead: // Set parameters
		IF ipModbusSlave[iLoopSlave].NumAddRegionRead <> 0 
		AND iLoopAdr <= (ipModbusSlave[iLoopSlave].NumAddRegionRead - 1) 
		THEN
			iQuantity := ipModbusSlave[iLoopSlave].AddressRead + ((iLoopAdr * 3 + 1) * SIZEOF(WORD));// arrAddressRead[iloopAdr][1] in Slave
			iMBAddr := ipModbusSlave[iLoopSlave].AddressRead + ((iLoopAdr * 3) * SIZEOF(WORD));// arrAddressRead[iloopAdr][0] in Slave
			UnitID := ipModbusSlave[iLoopSlave].UnitID;
			Quantity :=	iQuantity^;
			MBAddr := iMBAddr^;
			cbLength := SIZEOF(arrData);
			pMemoryAddr	:= ADR(arrData);
			peModbusFunction := ipModbusSlave[iLoopSlave].AddressRead + ((iLoopAdr * 3 + 2) * SIZEOF(WORD)); // arrAddressRead[iloopAdr][2] in Slave
			eModbusFunction := peModbusFunction^;
			iStepRunning := E_ModbusMasterStateRun.SendRequestRead;
		ELSE 
			iLoopAdr := 0;
			iStepRunning := E_ModbusMasterStateRun.ReturnReadDone;
		END_IF

			
	E_ModbusMasterStateRun.SendRequestRead: // Send request
		CASE eModbusFunction OF
			E_ModbusFunction.ReadHoldingRegisters:
				fbModbusMaster.ReadRegs(
					UnitID:= UnitID, 
					Quantity:= Quantity, 
					MBAddr:= MBAddr, 
					cbLength:= cbLength, 
					pMemoryAddr:= pMemoryAddr, 
					Execute:= TRUE,
					Timeout:= UINT_TO_TIME(iTimeout),
					BUSY=> bBusy, 
					Error=> bError , 
					ErrorId=>iErrorId 
				);
			
			E_ModbusFunction.ReadInputRegisters:
				fbModbusMaster.ReadInputRegs(
					UnitID:= UnitID, 
					Quantity:= Quantity, 
					MBAddr:= MBAddr, 
					cbLength:= cbLength, 
					pMemoryAddr:= pMemoryAddr, 
					Execute:= TRUE,
					Timeout:= UINT_TO_TIME(iTimeout),
					BUSY=> bBusy, 
					Error=> bError , 
					ErrorId=>iErrorId 
				);
			
		END_CASE
		iStepRunning := E_ModbusMasterStateRun.WaitReadRespond;
						
	E_ModbusMasterStateRun.WaitReadRespond:
		fbModbusMaster.ReadRegs(Execute := FALSE);
		fbModbusMaster.ReadInputRegs(Execute := FALSE);
		ipModbusSlave[iLoopSlave].ModbusErrorID := iErrorID;
		IF NOT fbModbusMaster.BUSY AND NOT fbModbusMaster.Error THEN
			iStepRunning := E_ModbusMasterStateRun.ConvertRawData;
			nNumberFaultRW := 0;
		END_IF
		
		IF fbModbusMaster.Error AND NOT fbModbusMaster.BUSY THEN
			iStepRunning := E_ModbusMasterStateRun.ReturnReadDone;
		END_IF
	
	E_ModbusMasterStateRun.ConvertRawData: 
		ipModbusSlave[iLoopSlave].Convert(
			iRegionNo := iLoopAdr,
		 	pReadData := ADR(arrData)
		);
		iLoopAdr := iLoopAdr + 1;
		iStepRunning := E_ModbusMasterStateRun.CheckNumberSlaveRegistered;

	E_ModbusMasterStateRun.ReturnReadDone: // Return, done
		iStepRunning := E_ModbusMasterStateRun.SetParametersWrite;
		iLoopAdr := 0;

	E_ModbusMasterStateRun.SetParametersWrite :
		IF  ipModbusSlave[iLoopSlave].NumAddRegionWrite <> 0
		AND iLoopAdr <= ipModbusSlave[iLoopSlave].NumAddRegionWrite - 1 
		THEN // iLoopAdr start from 1
			iMBAddr := ipModbusSlave[iLoopSlave].AddressWrite + (iLoopAdr * 11 * SIZEOF(WORD));// return address word contain value address( modbus) 
			pDataWrite := ipModbusSlave[iLoopSlave].AddressWrite + ((iLoopAdr * 11 + 2) * SIZEOF(WORD));
			iQuantity := ipModbusSlave[iLoopSlave].AddressWrite + ((iLoopAdr * 11 + 1) * SIZEOF(WORD));
			peModbusFunction := ipModbusSlave[iLoopSlave].AddressWrite + ((iLoopAdr * 11 + 10) * SIZEOF(WORD));
			eModbusFunction := peModbusFunction^;
			UnitID 	:=		ipModbusSlave[iLoopSlave].UnitID;
			Quantity	:=	iQuantity^;
			MBAddr	:=		iMBAddr^;
			cbLength	:= 	Quantity * 2;
			pMemoryAddr	:= 	pDataWrite;
			iStepRunning := E_ModbusMasterStateRun.SendRequestWrite;
		ELSE 
			iStepRunning := E_ModbusMasterStateRun.ReturnWriteDone;
		END_IF

	E_ModbusMasterStateRun.SendRequestWrite :
		CASE eModbusFunction OF
			E_ModbusFunction.WriteMultipleCoils:
				fbModbusMaster.WriteMultipleCoils(
					UnitID:= UnitID, 
					Quantity:= Quantity, 
					MBAddr:= MBAddr, 
					cbLength:= cbLength, 
					pMemoryAddr:= pMemoryAddr, 
					Execute:=  true,
					Timeout:= 	UINT_TO_TIME(iTimeout),	
					BUSY=> bBusy, 
					Error=> bError , 
					ErrorId=>iErrorId 
				);
													
			E_ModbusFunction.WriteMultipleRegisters:
				fbModbusMaster.WriteRegs(
					UnitID:= UnitID, 
					Quantity:= Quantity, 
					MBAddr:= MBAddr, 
					cbLength:= cbLength, 
					pMemoryAddr:= pMemoryAddr, 
					Execute:= TRUE,
					Timeout:= UINT_TO_TIME(iTimeout),	
					BUSY=> bBusy, 
					Error=> bError , 
					ErrorId=>iErrorId 
				);
											
			E_ModbusFunction.WriteSingleCoil:
				fbModbusMaster.WriteSingleCoil(
					UnitID:= UnitID, 
					Quantity:= Quantity, 
					MBAddr:= MBAddr, 
					cbLength:= cbLength, 
					pMemoryAddr:= pMemoryAddr, 
					Execute:=  true,
					Timeout:= UINT_TO_TIME(iTimeout),	
					BUSY=> bBusy, 
					Error=> bError , 
					ErrorId=>iErrorId 
				);
			E_ModbusFunction.WriteSingleRegister:
				fbModbusMaster.WriteSingleRegister(
					UnitID:= UnitID, 
					Quantity:= Quantity, 
					MBAddr:= MBAddr, 
					cbLength:= cbLength, 
					pMemoryAddr:= pMemoryAddr, 
					Execute:=  true,
					Timeout:= 	UINT_TO_TIME(iTimeout),	
					BUSY=> bBusy, 
					Error=> bError , 
					ErrorId=>iErrorId 
				);
		END_CASE
		
		iStepRunning := E_ModbusMasterStateRun.WaitWriteRespond;
	
	E_ModbusMasterStateRun.WaitWriteRespond :
		fbModbusMaster.WriteMultipleCoils( Execute := FALSE);
		fbModbusMaster.WriteRegs( Execute := FALSE);
		fbModbusMaster.WriteSingleCoil( Execute := FALSE);	
		fbModbusMaster.WriteSingleRegister( Execute := FALSE);
		ipModbusSlave[iLoopSlave].ModbusErrorID := iErrorID;
		IF NOT fbModbusMaster.BUSY AND NOT fbModbusMaster.Error THEN
			iStepRunning := E_ModbusMasterStateRun.SetParametersWrite;
			nNumberFaultRW := 0;
			iLoopAdr := iLoopAdr + 1;
		END_IF
		IF fbModbusMaster.Error AND NOT fbModbusMaster.BUSY THEN
			iStepRunning := E_ModbusMasterStateRun.ReturnWriteDone ;
		END_IF
	
	 E_ModbusMasterStateRun.ReturnWriteDone :
		iLoopAdr := 0;
		iLoopSlave := iLoopSlave + 1;// next slave
		IF iLoopSlave > iAmountSlave THEN
			iLoopSlave := 1;
		END_IF
		THIS^.tCalculateTimeRW(in := FALSE);
		tCalculateTimeRW(in := TRUE);
		iStepRunning := E_ModbusMasterStateRun.CheckNumberSlaveRegistered;
		
END_CASE
END_METHOD

METHOD protected StateStopping : BOOL (* Unit is uninitialized*)
iStepGeneral	:= E_ModBusMasterState.Uninitialized;
iStepRunning	:= E_ModbusMasterStateRun.notKnow;

iLoopSlave		:= 1;
iLoopAdr		:= 0;

fbModbusMaster(Execute := FALSE);
END_METHOD

METHOD protected StateStoppingDone : BOOL (* Unit is uninitialized*)
IF NOT bStop THEN
	iStepGeneral := E_ModBusMasterState.Ready;
END_IF
END_METHOD

METHOD protected StateUninitialized : BOOL (* Unit is uninitialized*)
END_METHOD

METHOD protected Stop : BOOL
IF iStepGeneral >= E_ModBusMasterState.Running AND iStepGeneral < E_ModBusMasterState.stop THEN
	iStepGeneral := E_ModBusMasterState.stop;
END_IF
bStop := TRUE;

Stop := (iStepGeneral = E_ModBusMasterState.stop_done);
END_METHOD

PROPERTY Timeout : UINT // in milisecond, if not respond in this time , error will raise
GET
Timeout := iTimeout;
END_GET
SET
iTimeout := Timeout;
END_SET
END_PROPERTY

END_FUNCTION_BLOCK

// ---- POUs/VFD/FB_VFD_ABB_ACS480.TcPOU
FUNCTION_BLOCK FB_VFD_ABB_ACS480 EXTENDS FB_UniversalVFDModbus

VAR
	VFD_CTRL_RUN_EMERGENCY_STOP : WORD;
	TempData0: U_Word2Int;
END_VAR

SUPER^();

METHOD Convert : BOOL
VAR_INPUT
	iRegionNo	:	INT;
	pReadData	:	POINTER TO word;
END_VAR
CASE	iRegionNo OF

	0: // status
		IF pReadData[0].15 = TRUE THEN
			eVfdStatus := VFD_STATUS_FAULT;
			
		ELSIF (eVfdState = VFD_INITIALIZING
			OR eVfdState = VFD_READY_INITIALIZED)
			AND pReadData[0].0 = TRUE
			AND pReadData[0].1 = TRUE	
			AND pReadData[0].2 = TRUE
			THEN
			eVfdStatus :=  VFD_STATUS_READY_TO_RUN;
				
		ELSIF pReadData[0].3 = FALSE THEN
			eVfdStatus :=  VFD_STATUS_STOP;
			
		ELSIF pReadData[0].3 = TRUE	//run
			AND pReadData[0].10 = FALSE	// Drive reference is in the forward direction	
			AND pReadData[0].11 = FALSE//Drive is running in the forward direction
			THEN		
			eVfdStatus := VFD_STATUS_RUNNING_FORWARD;
		
		ELSIF pReadData[0].3 = TRUE	//run
			AND pReadData[0].10 = TRUE	// Drive reference is in the forward direction	
			AND pReadData[0].11 = TRUE//Drive is running in the forward direction
			THEN		
			eVfdStatus := VFD_STATUS_RUNNING_REVERSE;
		
		END_IF
	1: 
		TempData0.iWord := pReadData[0];
		lrHzActual		:= ABS(INT_TO_LREAL( TempData0.iInt)*0.0025);//50/20000;	
		lrCurrent		:= WORD_TO_LREAL( pReadData[1])*0.01;	//46.05 = 100
		lrDcVoltage		:= WORD_TO_LREAL( pReadData[5])*0.1;	
	
	2: 
		lrVacOutToMotor	:= WORD_TO_LREAL( pReadData[0]);	//4099	/1
		lrPowerKw		:= WORD_TO_LREAL( pReadData[1])*0.01;		//46.04
	
	3:
		lrTotalKwh :=  WORD_TO_LREAL( pReadData[0])*0.1;
		
	4: 
		lrSpeed :=  WORD_TO_LREAL( pReadData[0]);
	
	


END_CASE
END_METHOD

METHOD  FirstCycle 
VAR_INPUT
	sName : STRING;
	iUnitID : BYTE ; // modbus address of the device : 1- 255
END_VAR
SUPER^.FirstCycle( sName := sName, iUnitID := iUnitID);
(*Assign Ctrol Word : user Manual M-driver*)
VFD_CTRL_RESET_FAULT := 2#0001_0001;
VFD_CTRL_RUN_FORWARD := 2#0000_0010;
VFD_CTRL_RUN_REVERSE := 2#0000_0110;
VFD_CTRL_STOP_FREE 	 := 2#0010_0000_0001;
VFD_CTRL_STOP_SPEED_DOWN := 2#1000_0001;
VFD_CTRL_RUN_EMERGENCY_STOP := 2#0001_0000_0001;

// actual state	
	arrAddressRead[0][0] := 3;
	arrAddressRead[0][1] := 1;
	arrAddressRead[0][2] := E_ModbusFunction.ReadHoldingRegisters;

//mode0 address = 40000 + function*100 + sub function -1
	// actual hz  
	arrAddressRead[1][0] := 105; // 01.06
	arrAddressRead[1][1] := 6;
	arrAddressRead[1][2] := E_ModbusFunction.ReadHoldingRegisters;
	
	arrAddressRead[2][0] := 112; // 01.13
	arrAddressRead[2][1] := 2;
	arrAddressRead[2][2] := E_ModbusFunction.ReadHoldingRegisters;
	
	arrAddressRead[3][0] := 119; // 01.20
	arrAddressRead[3][1] := 1;
	arrAddressRead[3][2] := E_ModbusFunction.ReadHoldingRegisters;
	
	arrAddressRead[4][0] := 101; // 01.20
	arrAddressRead[4][1] := 1;
	arrAddressRead[4][2] := E_ModbusFunction.ReadHoldingRegisters;
iNumAddRegionRead	:= 5;

/////write control WORD VFD, // use ctrol word and frequency in 1 modbus write
arrAddressWrite[iCTRL_WORD][0]	:= 0;
arrAddressWrite[iCTRL_WORD][1]	:= 2;
arrAddressWrite[iCTRL_WORD][2]	:= VFD_CTRL_STOP_FREE;
arrAddressWrite[iCTRL_WORD][10]	:= E_ModbusFunction.WriteMultipleRegisters;

// Frequency
//arrAddressWrite[iCTRL_FREQUENCY_WORD][0]	:= 1;
//arrAddressWrite[iCTRL_FREQUENCY_WORD][1]	:= 1;
							(*MUST BE CARE FULL WHEN USE FLOATING POINT CONVERT*)
arrAddressWrite[iCTRL_FREQUENCY_WORD][3]	:= LREAL_TO_WORD( FC_ScaleValue(	rangeRawMin := 0,
																				rangeRawMax := 50,
																				RangeScaleMin :=0,
																				RangeScaleMax := 20000,
																				ValueRaw := 0)
										  );
										  
iNumAddRegionWrite := 1;// use ctrol word and frequency in 1 modbus write

bSwap	:= TRUE;
END_METHOD

METHOD PROTECTED  MS_Aborting
arrAddressWrite[iCTRL_WORD][2]	:= VFD_CTRL_STOP_FREE;
SUPER^.MS_Aborting();
END_METHOD

METHOD  PROTECTED  MS_Initializing
SUPER^.MS_Initializing();
END_METHOD

METHOD PROTECTED  MS_RunForward
VAR_INPUT
END_VAR
// use ctrol word and frequency in 1 modbus write WRITE MULTIES REGIS
arrAddressWrite[iCTRL_WORD][3] :=  LREAL_TO_WORD( 
															FC_ScaleValue(	rangeRawMin := 0,
																			rangeRawMax := 50,
																			RangeScaleMin := 0,
																			RangeScaleMax := 20000,
																			ValueRaw := lrHzControl) 
																				);
SUPER^.MS_RunForward();
END_METHOD

METHOD PROTECTED  MS_RunReverse
VAR_INPUT
END_VAR
// use ctrol word and frequency in 1 modbus write WRITE MULTIES REGIS
arrAddressWrite[iCTRL_WORD][3] :=  LREAL_TO_WORD( 
															FC_ScaleValue(	rangeRawMin := 0,
																			rangeRawMax := 50,
																			RangeScaleMin := 0,
																			RangeScaleMax := 20000,
																			ValueRaw := lrHzControl) 
																				);
SUPER^.MS_RunReverse();
END_METHOD

END_FUNCTION_BLOCK

// ---- POUs/VFD/FB_UniversalVFDModbus.TcPOU
FUNCTION_BLOCK abstract FB_UniversalVFDModbus EXTENDS FB_ModbusSlave IMPLEMENTS I_UniversalVFD
VAR
	eVfdState	: E_Vfd_State;
	bInit	: BOOL;
	bBusy	: BOOL;
	bReset	: BOOL;
	bStop	: BOOL;
	bAbort : BOOL;
	bError : BOOL;
	bWarning : BOOL;// status
	bRunningForward	: BOOL;// in state running forward
	bRunningReverse	: BOOL; // in state running reverse
	bRanForward	: BOOL;
	bRanReverse	: BOOL;
	lrHzActual	: LREAL;
	lrDcVoltage		: LREAL;
	lrVacOutToMotor	: LREAL;
	lrCurrent	: LREAL;	
	lrPowerKw	: LREAL;	
	eVfdStatus	: E_VFD_Status;
	lrHzControl	: LREAL;// value in range(0.0-50.0Hz)
	iErrorID		: UDINT;

	lrSpeed : LREAL;
	lrTorque : LREAL;
	lrTotalKwh : LREAL;
	lrRatedPower : LREAL;
	bActive: BOOL;
	bOverLoad: BOOL;
	bStopLog: BOOL;
	bStopped: BOOL;
	
	VFD_CTRL_RESET_FAULT : WORD;
	VFD_CTRL_RUN_FORWARD :WORD;
	VFD_CTRL_RUN_REVERSE :WORD ;
	VFD_CTRL_STOP_FREE 		:WORD ;
	VFD_CTRL_STOP_SPEED_DOWN	:WORD ;
	
	tonStopDelay: Ton;
	// time delay after status = stop
	tStopDelay: TIME := T#4S;

END_VAR
VAR CONSTANT
	// index
	iCTRL_WORD	: UINT := 1;
	iCTRL_FREQUENCY_WORD :UINT := 0;
	iSTATUS_WORD	: UINT := 0;


END_VAR

StateMachine();
CASE eVfdStatus OF
	VFD_STATUS_RUNNING_FORWARD :
		bRanForward := TRUE;
		bRanReverse := FALSE;
		bStopped := FALSE;
	VFD_STATUS_RUNNING_REVERSE:
		bRanForward := FALSE;
		bRanReverse := TRUE;
		bStopped := FALSE;
	VFD_STATUS_FAULT,VFD_STATUS_STOP:
		bRanForward := FALSE;
		bRanReverse := FALSE;
		bStopped := TRUE;
		
END_CASE
bError := eVfdStatus = VFD_STATUS_FAULT;
bActive := eVfdState >= VFD_IDLE;

{attribute 'monitoring' := 'variable'}
PROPERTY Active : REFERENCE TO  bool
GET
Active REF= bActive;
END_GET
END_PROPERTY

PROPERTY AcVoltageToMotor : Reference to lreal
GET
AcVoltageToMotor ref= lrVacOutToMotor;
END_GET
END_PROPERTY

{attribute 'monitoring' := 'variable'}
PROPERTY Busy : reference to bool
GET
Busy ref= bBusy;
END_GET
END_PROPERTY

METHOD Convert : BOOL
VAR_INPUT
	iRegionNo	:	INT;
	pReadData	:	POINTER TO word;
END_VAR
(*CASE iRegionNo OF
	0:
		// Status word
		Inverter_Ready		:=  pReadData[0].0;
		InverterReadyToRun	:=  pReadData[0].1;
		InverterRunning		:=  pReadData[0].2;
		InverterFaultActive :=  pReadData[0].3;
		OFF2_active			:= NOT pReadData[0].4;
		OFF3_active			:= NOT  pReadData[0].5;
		ON_inhibit_active 	 := pReadData[0].6;
		Inverter_warning_active := pReadData[0].7;
		Deviation_setpoint_OR_ActiveValue := NOT pReadData[0].8;
		PZD_control 		:= pReadData[0].9;
		Motor_current_Or_torque_limit  := NOT pReadData[0].11;
		Brake_open	 := pReadData[0].12;
		Motor_overload := NOT pReadData[0].13;
		Motor_RunRight	:= pReadData[0].14;
		Inverter_overload :=  NOT pReadData[0].15;
		
		IF InverterFaultActive THEN
			eStatus := VFD_STATUS_FAULT;
		ELSIF InverterFaultActive THEN
			eStatus := VFD_STATUS_WARNING;
		ELSIF InverterRunning THEN
			IF Motor_RunRight THEN
				eStatus := VFD_STATUS_RUNNING_FORWARD;
			ELSE
				eStatus := VFD_STATUS_RUNNING_REVERSE;
			END_IF
		ELSIF NOT InverterRunning THEN
			eStatus := VFD_STATUS_STOP;
		END_IF

		// Speed word
		lrHz_actual := WORD_TO_LREAL( pReadData[1])*50/16383;
		
	1:
		///  actual  Speed ( rpm) (unit A : Scale factor 1), Current ( A , 100, , Torque (Nm, 100)
	//, Actual Power (kw, 100), Total Kwh( 1), Dc bus Voltage(1), REFERENCE( hz, 100), RATED PWR( 100),OUTPUT VOLTS(1)
		lrSpeed := pReadData[0];
		lrCurrent := WORD_TO_LREAL(pReadData[1])/100;
		lrTorque := WORD_TO_LREAL(pReadData[2])/100;
		lrPower := WORD_TO_LREAL(pReadData[3])/100;
		lrTotalKwh := WORD_TO_LREAL(pReadData[4]);
		lrDc_Voltage := WORD_TO_LREAL(pReadData[5]);
		lrRatedPower := WORD_TO_LREAL(pReadData[7])/100;
		lrVAC_OutToMotor := WORD_TO_LREAL(pReadData[8]);
END_CASE
*)
END_METHOD

PROPERTY Current : reference to lreal
GET
Current ref= lrCurrent;
END_GET
END_PROPERTY

PROPERTY DcVoltage : Reference to lreal
GET
DcVoltage ref= lrDcVoltage;
END_GET
END_PROPERTY

{attribute 'monitoring' := 'variable'}
PROPERTY Error : REFERENCE to bool
GET
Error ref= bError;
END_GET
END_PROPERTY

{attribute 'monitoring' := 'variable'}
PROPERTY ErrorID : reference to UDINT
GET
ErrorID ref= iErrorID;
END_GET
END_PROPERTY

METHOD  FirstCycle 
VAR_INPUT
	sName : STRING;
	iUnitID : BYTE ; // modbus address of the device : 1- 255
END_VAR
THIS^.sName := sName;
THIS^.iUnitID := iUnitID;
(*(*HSW (speed setpoint), HIW (actual speed), STW (control word), ZSW (status word) refer to
control data. For more information, see parameters r2018 and P2019 in Chapter "Parameter
list (Page 147)*)
//ZSW  (status WORD), HIW (actual speed)
	arrAddress[0][0] := 109;
	arrAddress[0][1]	:= 2;

///  actual  Speed ( rpm) (unit A : Scale factor 1), Current ( A , 100, , Torque (Nm, 100)
	//, Actual Power (kw, 100), Total Kwh( 1), Dc bus Voltage(1), REFERENCE( hz, 100), RATED PWR( 100),OUTPUT VOLTS(1)
	arrAddress[1][0] := 24;
	arrAddress[1][1] := 10;

	
iNumAddRegion	:= 2;
/////write control  VFD
	
// Frequency

arrAddressWrite[0][0]	:= 100;
arrAddressWrite[0][1] 	:= 1;
arrAddressWrite[0][2]	:= LREAL_TO_WORD( FC_ScaleValue(	rangeRawMin := 0,
															rangeRawMax := 50,
															RangeScaleMin :=0,
															RangeScaleMax := 16384,
															ValueRaw := lrHz_Control) );
// Control word																	
arrAddressWrite[1][0]	:= 99;
arrAddressWrite[1][1] := 1;
arrAddressWrite[1][2]	:= 1150; //VFD_CTRL_STOP_SPEED_DOWN
iNumAddRegionWrite := 2;
*)
END_METHOD

PROPERTY HzActual : REFERENCE TO  LReal
GET
HzActual ref= lrHzActual;
END_GET
END_PROPERTY

PROPERTY HzControl : reference to LReal
GET
HzControl ref= lrHzControl;
END_GET
END_PROPERTY

{attribute 'monitoring' := 'variable'}
PROPERTY InHz : bool
GET
InHz :=  F_InRange( bound1 := lrHzControl +1,
					bound2 := lrHzControl -1,
					value := lrHzActual) ;
END_GET
END_PROPERTY

PROPERTY isRunForward : bool
GET
isRunForward := bRanForward;
END_GET
END_PROPERTY

{attribute 'monitoring' := 'variable'}
PROPERTY IsRunning : bool
GET
IsRunning := eVfdStatus = VFD_STATUS_RUNNING_FORWARD
			 OR  eVfdStatus = VFD_STATUS_RUNNING_REVERSE;
END_GET
END_PROPERTY

PROPERTY isRunReverse : bool
GET
isRunReverse := bRanReverse;
END_GET
END_PROPERTY

PROPERTY isStop : bool
GET
isStop := bStopped;
END_GET
END_PROPERTY

METHOD MR_Abort : BOOL
VAR_INPUT
END_VAR
IF eVfdState >= VFD_INITIALIZING THEN
	bAbort := TRUE;
	eVfdState := VFD_ABORTING;
	fbMachineLogger.MR_AddLogs(CONCAT(sName,' : abort requested'));
	bBusy := TRUE;
	
ELSIF eVfdState = VFD_UNINITIALIZED THEN
	bAbort 		:= FALSE;
	MR_Abort	:= TRUE;
	bBusy := FALSE;
	fbMachineLogger.MR_AddLogs(CONCAT(sName,' : abort done'));
	
END_IF
END_METHOD

METHOD MR_Init : bool
VAR_INPUT
END_VAR
IF eVFDState = VFD_UNINITIALIZED THEN
	bInit := TRUE;
	MR_Init := FALSE;
	eVfdState := VFD_INITIALIZING;
	fbMachineLogger.MR_AddLogs(CONCAT(sName,' : initialization requested'));
	bBusy := TRUE;
	
ELSIF eVFDState = VFD_READY_INITIALIZED THEN
	bInit := FALSE;
	MR_Init := TRUE;
	bBusy := FALSE;
	fbMachineLogger.MR_AddLogs(CONCAT(sName,' : initialization done'));
END_IF
END_METHOD

METHOD MR_Reset : BOOL
VAR_INPUT
END_VAR
IF eVfdState >= VFD_IDLE AND bError THEN
	bReset := TRUE;
	eVfdState := VFD_RESET;
	fbMachineLogger.MR_AddLogs(CONCAT(sName,' : reset requested'));			
	bBusy := TRUE;
	
ELSIF eVfdState = VFD_RESET_DONE THEN
	bError := FALSE;
	iErrorID := 0;
	bReset := FALSE;
	MR_Reset := TRUE;
	bBusy := FALSE;
	fbMachineLogger.MR_AddLogs(CONCAT(sName,' : reset done'));		
		
END_IF
END_METHOD

METHOD MR_RunForward : BOOL
VAR_INPUT
	hz : LREAL; 
END_VAR
IF eVfdState = VFD_IDLE  AND (NOT  F_InRange( 	bound1 := lrHzControl + 0.01,
												bound2 := lrHzControl - 0.01,
												value :=  hz)
								OR bRanReverse
								OR bStopped)
THEN
	lrHzControl := hz;
	bRunningForward := TRUE;
	MR_RunForward := FALSE;
	eVfdState := VFD_RUN_FORWARD;
	fbMachineLogger.MR_AddLogs( sLogMessage := FUN_MergeStrings4(  sName,' : run ',LREAL_TO_STRING( lrHzControl),' forward requested'));		
	bBusy := TRUE;
	
ELSIF eVfdState = VFD_RUN_FORWARD_DONE THEN
	bRunningForward := FALSE;
	MR_RunForward := TRUE;
	fbMachineLogger.MR_AddLogs(CONCAT(sName,' : run forward done'));	
	bBusy := FALSE;
END_IF
END_METHOD

METHOD MR_RunReverse : BOOL// must stop before call run reverse or forward
VAR_INPUT
	hz : LREAL; // >0 and < 50;
END_VAR
IF eVfdState = VFD_IDLE  AND (NOT  F_InRange( 	bound1 := lrHzControl + 0.01,
												bound2 := lrHzControl - 0.01,
												value :=  hz)
								OR bRanForward
								OR bStopped)
THEN
	lrHzControl := hz;
	bRunningReverse := TRUE;
	MR_RunReverse := FALSE;
	eVfdState := VFD_RUN_REVERSE;
	fbMachineLogger.MR_AddLogs( sLogMessage := FUN_MergeStrings4(  sName,' : run ',LREAL_TO_STRING( lrHzControl),' forward requested'));		
	bBusy := TRUE;
	
ELSIF eVfdState = VFD_RUN_REVERSE_DONE THEN
	bRunningReverse := FALSE;
	MR_RunReverse := TRUE;
	fbMachineLogger.MR_AddLogs(CONCAT(sName,' : run forward done'));
	bBusy := FALSE;
END_IF
END_METHOD

METHOD MR_Stop : BOOL
VAR_INPUT
END_VAR
IF eVfdState >= VFD_IDLE AND eVfdState <> VFD_STOP_DONE THEN
	IF NOT bStopLog THEN 
		fbMachineLogger.MR_AddLogs(CONCAT(sName,' : stop requested'));
		bStopLog := TRUE;	
	END_IF
	
	bStop := TRUE;
	eVfdState := VFD_STOP;
	bBusy := TRUE;
	
ELSIF eVfdState = VFD_STOP_DONE THEN
	bStop 		:= FALSE;
	MR_Stop 	:= TRUE;
	bStopLog 	:= FALSE;
	fbMachineLogger.MR_AddLogs(CONCAT(sName,' : stop done'));	
	bBusy := FALSE;
END_IF
END_METHOD

METHOD PROTECTED MS_Aborting
lrHzControl := 0;
bInit := FALSE;
bRunningForward := FALSE;
bRunningReverse := FALSE;
bReset := FALSE;
bRanForward := FALSE;
bRanReverse := FALSE;
bOverLoad := FALSE;
bStop := FALSE;
bStopLog := FALSE;
bStopped := FALSE;
THIS^.tonStopDelay(IN :=FALSE);
IF eVfdStatus = VFD_STATUS_STOP OR eVfdStatus = VFD_STATUS_FAULT THEN
	eVfdState := VFD_UNINITIALIZED;
END_IF
END_METHOD

METHOD PROTECTED MS_Idle
;
END_METHOD

METHOD  PROTECTED  MS_Initializing
// from Subclass call Super^.MS_Initializing
arrAddressWrite[iCTRL_WORD][2]	:= VFD_CTRL_RESET_FAULT;
IF eVfdStatus = VFD_STATUS_READY_TO_RUN THEN
	eVFDState := VFD_READY_INITIALIZED;
END_IF
END_METHOD

METHOD PROTECTED MS_ReadyInitialized
VAR_INPUT
END_VAR
IF NOT bInit THEN
	eVfdState := VFD_IDLE;
END_IF
END_METHOD

METHOD PROTECTED  MS_Reset
VAR_INPUT
END_VAR
arrAddressWrite[iCTRL_WORD][2]	:= VFD_CTRL_RESET_FAULT;
IF THIS^.evfdStatus <>  VFD_STATUS_NOT_RESPOND AND
	THIS^.evfdStatus <>  VFD_STATUS_FAULT THEN
	evfdState := VFD_RESET_DONE;
END_IF
END_METHOD

METHOD PROTECTED MS_ResetDone
VAR_INPUT
END_VAR
IF NOT bReset THEN
	evfdState := VFD_IDLE;
END_IF
END_METHOD

METHOD PROTECTED  MS_RunForward
VAR_INPUT
END_VAR
(*arrAddressWrite[iCtrlFrequencyWord][2] :=  LREAL_TO_WORD( 
											FC_ScaleValue(		rangeRawMin := 0,
																rangeRawMax := 50,
																RangeScaleMin := WORD_TO_LREAL( wHzWordValueMin),
																RangeScaleMax := WORD_TO_LREAL( wHzWordValueMax),
																ValueRaw := lrHzControl) 
														);*)
arrAddressWrite[iCTRL_WORD][2]	:= VFD_CTRL_RUN_FORWARD;
IF eVfdStatus = VFD_STATUS_RUNNING_FORWARD 
(*AND F_InRange( bound1 := lrHzControl + 1,
				bound2 := lrHzControl -1,
				value := lrHzActual)*)
THEN
	eVFDState := VFD_RUN_FORWARD_DONE;
END_IF
END_METHOD

METHOD PROTECTED MS_RunForwardDone
IF NOT bRunningForward THEN
	eVfdState := VFD_IDLE;
END_IF
END_METHOD

METHOD PROTECTED  MS_RunReverse
VAR_INPUT
END_VAR
(*arrAddressWrite[iCtrlFrequencyWord][2] :=  LREAL_TO_WORD( 
											FC_ScaleValue(		rangeRawMin := 0,
																rangeRawMax := 50,
																RangeScaleMin := WORD_TO_LREAL( wHzWordValueMin),
																RangeScaleMax := WORD_TO_LREAL( wHzWordValueMax),
																ValueRaw := lrHzControl) 
														);*)
arrAddressWrite[iCTRL_WORD][2]	:= VFD_CTRL_RUN_REVERSE;
IF eVfdStatus = VFD_STATUS_RUNNING_REVERSE 
(*AND F_InRange( bound1 := lrHzControl + 1,
				bound2 := lrHzControl -1,
				value := lrHzActual)*)
THEN
	eVFDState := VFD_RUN_REVERSE_DONE;
END_IF
END_METHOD

METHOD PROTECTED MS_RunReverseDone
VAR_INPUT
END_VAR
IF NOT bRunningReverse THEN
	eVfdState := VFD_IDLE;
END_IF
END_METHOD

METHOD protected  MS_Stop 
VAR_INPUT
END_VAR
arrAddressWrite[iCTRL_WORD][2]	:= VFD_CTRL_STOP_SPEED_DOWN;
(*tonStopDelay( in := eVfdStatus = VFD_STATUS_STOP,
				PT := tStopDelay);*)
IF eVfdStatus = VFD_STATUS_STOP THEN
 eVfdState := VFD_STOP_DONE;	
END_IF
(*IF tonStopDelay.Q THEN
	tonStopDelay(IN := FALSE);
	
END_IF*)
END_METHOD

METHOD protected Ms_StopDone
VAR_INPUT
END_VAR
IF NOT bStop THEN
	eVfdState := VFD_IDLE;
END_IF
END_METHOD

METHOD PROTECTED MS_Uninitialized
END_METHOD

{attribute 'monitoring' := 'variable'}
PROPERTY Overload : reference TO BOOL
GET
Overload REF= bOverLoad;
END_GET
END_PROPERTY

{attribute 'monitoring' := 'variable'}
PROPERTY PowerKw : REFERENCE TO LREAL
GET
PowerKw ref= lrPowerKw;
END_GET
END_PROPERTY

PROPERTY Speed : Reference to lreal
GET
Speed REF= lrSpeed;
END_GET
END_PROPERTY

{attribute 'monitoring' := 'variable'}
PROPERTY State : reference to E_Vfd_State
GET
State REF= eVfdState;
END_GET
END_PROPERTY

METHOD PROTECTED StateMachine
CASE eVfdState OF
	VFD_UNINITIALIZED :
		MS_Uninitialized();
		
	VFD_INITIALIZING	:
		MS_Initializing();
		
	VFD_READY_INITIALIZED :
		MS_ReadyInitialized();
		
	VFD_IDLE:
		MS_Idle();
	
	VFD_RUN_FORWARD	:
		MS_RunForward();
		
	VFD_RUN_FORWARD_DONE:
		MS_RunForwardDone();
	
	VFD_RUN_REVERSE	:
		MS_RunReverse();
	
	VFD_RUN_REVERSE_DONE:
		MS_RunReverseDone();
	
	VFD_STOP		:
		MS_Stop();
		
	VFD_STOP_DONE	:
		Ms_StopDone();
		
	VFD_RESET	:
		MS_Reset();
		
	VFD_RESET_DONE	:
		MS_ResetDone();
		
	VFD_ABORTING :
		MS_Aborting();
	
	
END_CASE
END_METHOD

{attribute 'monitoring' := 'variable'}
PROPERTY Status : reference to E_VFD_Status
GET
Status REF= eVfdStatus;
END_GET
END_PROPERTY

PROPERTY timeStopDelay : time
GET
timeStopDelay := THIS^.tStopDelay;
END_GET
SET
tStopDelay := timeStopDelay;
END_SET
END_PROPERTY

PROPERTY Torque : reference to lreal
GET
Torque ref= Torque;
END_GET
END_PROPERTY

PROPERTY TotalKwh : reference to lreal
GET
TotalKwh REF= TotalKwh;
END_GET
END_PROPERTY

// not all vfd modbus available this function 
PROPERTY Warning : reference to bool
GET
Warning  ref= bWarning;
END_GET
END_PROPERTY

END_FUNCTION_BLOCK

// ---- POUs/VFD/FB_VFD_Mdriver.TcPOU
FUNCTION_BLOCK FB_VFD_Mdriver EXTENDS FB_UniversalVFDModbus

VAR
	eFaultInfor	: E_VfdMdriverFaultInfor;
END_VAR

//bError := eVfdStatus
SUPER^();

METHOD Convert : BOOL
VAR_INPUT
	iRegionNo	:	INT;
	pReadData	:	POINTER TO word;
END_VAR
CASE	iRegionNo OF
	0: 
	
		lrHzActual		:= WORD_TO_LREAL( pReadData[0])*0.01;	//4097	/unit /100
		lrDcVoltage		:= WORD_TO_LREAL( pReadData[1])*0.1;	//4098 	/10
		lrVacOutToMotor	:= WORD_TO_LREAL( pReadData[2]);	//4099	/1
		lrCurrent		:= WORD_TO_LREAL(  pReadData[3])*0.01;		//4100	/100
		//4 reserve
		lrPowerKw		:= WORD_TO_LREAL(  pReadData[5])*0.001;		//4102	/1000> kW
	
	1: // status
		CASE pReadData[0] OF
			0: eVfdStatus := VFD_STATUS_STOP;
			
			1: 
				eVfdStatus := VFD_STATUS_RUNNING_FORWARD;
			2:
				eVfdStatus := VFD_STATUS_RUNNING_REVERSE;
			3: 
				eVfdStatus := VFD_STATUS_STOP;
		END_CASE
		// important
		IF eVfdState = VFD_INITIALIZING THEN
			IF eFaultInfor = E_VfdMdriverFaultInfor.Nofault
			AND eVfdStatus = VFD_STATUS_STOP THEN
				eVfdStatus := VFD_STATUS_READY_TO_RUN;
			ELSIF eFaultInfor <> E_VfdMdriverFaultInfor.Nofault THEN
				eVfdStatus := VFD_STATUS_FAULT;
			END_IF
		END_IF
		IF eFaultInfor <> E_VfdMdriverFaultInfor.Nofault THEN
			eVfdStatus := VFD_STATUS_FAULT;
		END_IF
		IF iModbusErrorID = MODBUSERROR_NO_RESPONSE THEN
			eVfdStatus := VFD_STATUS_NOT_RESPOND;
		END_IF
		// important
	
	2: 
	
		iErrorID := WORD_TO_UDINT( pReadData[0]);
		eFaultInfor :=  WORD_TO_UINT( pReadData[0]);
END_CASE
END_METHOD

METHOD  FirstCycle 
VAR_INPUT
	sName : STRING;
	iUnitID : BYTE ; // modbus address of the device : 1- 255
END_VAR
SUPER^.FirstCycle( sName := sName, iUnitID := iUnitID);
(*Assign Ctrol Word : user Manual M-driver*)
VFD_CTRL_RESET_FAULT := 7;
VFD_CTRL_RUN_FORWARD := 1;
VFD_CTRL_RUN_REVERSE := 2;
VFD_CTRL_STOP_FREE 		:= 5;
VFD_CTRL_STOP_SPEED_DOWN	:= 6;
///  actual hz, current, voltage
arrAddressRead[0][0] := 4097;
arrAddressRead[0][1]	:= 6;
arrAddressRead[0][2]	:= E_ModbusFunction.ReadHoldingRegisters;

// actual state	
arrAddressRead[1][0] := 16#3000;
arrAddressRead[1][1]	:= 1;
arrAddressRead[1][2]	:= E_ModbusFunction.ReadHoldingRegisters;

// fault infor
arrAddressRead[2][0] := 16#8000;
arrAddressRead[2][1]	:= 1;
arrAddressRead[2][2]	:= E_ModbusFunction.ReadHoldingRegisters;

iNumAddRegionRead	:= 3;

/////write control WORD VFD
arrAddressWrite[iCTRL_WORD][0]	:= 16#2000;
arrAddressWrite[iCTRL_WORD][1]	:= 1;
arrAddressWrite[iCTRL_WORD][2]	:= VFD_CTRL_STOP_FREE;
arrAddressWrite[iCTRL_WORD][10]	:= E_ModbusFunction.WriteSingleRegister;
// Frequency
arrAddressWrite[iCTRL_FREQUENCY_WORD][0]	:= 4096;
arrAddressWrite[iCTRL_FREQUENCY_WORD][1]	:= 1;
							(*MUST BE CARE FULL WHEN USE FLOATING POINT CONVERT*)
arrAddressWrite[iCTRL_FREQUENCY_WORD][2]	:= LREAL_TO_WORD( FC_ScaleValue(	rangeRawMin := 0,
															rangeRawMax := 50,
															RangeScaleMin :=0,
															RangeScaleMax := 10000,
															ValueRaw := 0)
										  );
arrAddressWrite[iCTRL_FREQUENCY_WORD][10]	:= E_ModbusFunction.WriteSingleRegister;
										  
iNumAddRegionWrite := 2;

bSwap	:= TRUE;
END_METHOD

METHOD PROTECTED  MS_Aborting
arrAddressWrite[iCTRL_WORD][2]	:= VFD_CTRL_STOP_FREE;
SUPER^.MS_Aborting();
END_METHOD

METHOD PROTECTED  MS_RunForward
VAR_INPUT
END_VAR
arrAddressWrite[iCTRL_FREQUENCY_WORD][2] :=  LREAL_TO_WORD( 
															FC_ScaleValue(	rangeRawMin := 0,
																			rangeRawMax := 50,
																			RangeScaleMin := 0,
																			RangeScaleMax := 10000,
																			ValueRaw := lrHzControl) 
																				);
SUPER^.MS_RunForward();
END_METHOD

METHOD PROTECTED  MS_RunReverse
VAR_INPUT
END_VAR
arrAddressWrite[iCTRL_FREQUENCY_WORD][2] :=  LREAL_TO_WORD( 
															FC_ScaleValue(	rangeRawMin := 0,
																			rangeRawMax := 50,
																			RangeScaleMin := 0,
																			RangeScaleMax := 10000,
																			ValueRaw := lrHzControl) 
																				);
SUPER^.MS_RunReverse();
END_METHOD

END_FUNCTION_BLOCK

// ---- TEST/FB_ModbusMaster_Test.TcPOU
(* FB relate to Hardware *)
FUNCTION_BLOCK FB_ModbusMaster_Test EXTENDS FB_TestSuite
VAR
END_VAR

END_FUNCTION_BLOCK

// ---- TEST/FB_ModbusSlave_Test.TcPOU
FUNCTION_BLOCK FB_ModbusSlave_Test EXTENDS FB_TestSuite
VAR
END_VAR

END_FUNCTION_BLOCK

// ---- TEST/FB_UniversalVFDModbus_Ex.TcPOU
FUNCTION_BLOCK FB_UniversalVFDModbus_Ex EXTENDS FB_UniversalVFDModbus

SUPER^();

METHOD Convert : BOOL
VAR_INPUT
	iRegionNo	:	INT;
	pReadData	:	POINTER TO word;
END_VAR
CASE iRegionNo OF
	0:
		IF pReadData[0] = 10 THEN
			eVfdStatus := VFD_STATUS_READY_TO_RUN;
		END_IF
END_CASE
END_METHOD

END_FUNCTION_BLOCK

// ---- TEST/FB_UniversalVFDModbus_Test.TcPOU
FUNCTION_BLOCK FB_UniversalVFDModbus_Test EXTENDS FB_TestSuite

VAR
	FbVFDModbus : FB_UniversalVFDModbus_Ex;
	nCycle	: ULINT;
	tonBetweenTestCase		: TON;
	tBetweenTestCase		: TON;
	indexTestCase			: UDINT; // +1 each test case
	arrDataRead				: ARRAY [0..50] OF WORD; 
END_VAR
VAR
	STATUS_NOT_RESPOND		:WORD :=  0;
	STATUS_READY_TO_RUN		:WORD:= 1;
	STATUS_STOP				:WORD:= 2;
	STATUS_RUNNING_FORWARD	:WORD:= 3;
	STATUS_RUNNING_REVERSE	:WORD:= 4;
	STATUS_WARNING			:WORD:= 6;// should not use
	STATUS_FAULT			:WORD:= 7;
END_VAR
//for Intergrate Test// if want to test any FB extent FB_UniversalVFDModbus => replace the FB_UniversalVFDModbus_Ex.

WhenFirstCycleExpectNameAndUinitIDTheSame();//Cycle 0
WhenUnInitializedExpect_Active_Busy_areFalse();//Cycle 0
WhenUnInitializedMR_InitExpectStateInitializing();//Cycle 0
WhenInitializingExpectActiveFalseAndBusyTrue();//Cycle 0
WhenInitializingAndStatusReadyToRunExpectStateReadyInitialized(nThCycle := 1, nCycleDuration := 2);
WhenStateAlreadyInitializedAndCallMR_initExpectStateIsVFD_IDLE(nThCycle := 3, nCycleDuration := 2);
WhenIdleAndIsStopCallMr_RunForwardExpectVFD_Run_Forward( nThCycle := 5, nCycleDuration := 1);
WhenVFD_RUN_FORWARDAndVFD_STATUS_RUNFORWARDExpectVFD_RUNFORWARD_DONE(nThCycle := 6, nCycleDuration := 1);
nCycle := nCycle +1 ;

FbVFDModbus();

METHOD protected WhenFirstCycleExpectNameAndUinitIDTheSame
VAR	
		sNameResult	: STRING;
		iUinitIDResult	: BYTE;
	// @TEST-FIXTURE Also as @TEST-EXPECT
		sName_In : STRING := 'VFD';
		iUinitID_In : BYTE := 43;
END_VAR
TEST( 'When Set Name expect ');

// @TEST-RUN
FbVFDModbus.FirstCycle( sName := sName_In,
						iUnitID := iUinitID_In);
	
sNameResult := FbVFDModbus.Name;
iUinitIDResult := FbVFDModbus.UnitID;				
// @TEST-ASSERT
AssertEquals( Expected := sName_In,
				Actual := sNameResult,
				Message := 'Test Set name Fail');
				
AssertEquals( Expected := iUinitID_In,
				Actual := iUinitIDResult,
				Message := 'Test Set Id Address Fail');
				
// always Remember Implement Test_finished	
TEST_FINISHED();
indexTestCase := 1;
END_METHOD

METHOD PROTECTED WhenIdleAndIsStopCallMr_RunForwardExpectVFD_Run_Forward
VAR_INPUT
	nThCycle : ULINT;// the cycle call implement
	nCycleDuration : UINT := 1;// number cycle this method be called
END_VAR
VAR
	bIsStopACT : BOOL;
	bActiveACT : BOOL;
	bBusyACT	: BOOL;
	eStateACT : E_VFD_State;
	eStatusACT	: E_VFD_Status;
	//@TEST-FIXTURE
	eStateFixture	: E_VFD_State := VFD_IDLE;
	bIsStopFixture	: BOOL := true;
	//@TEST-EXPECT
	eStateExp	: E_VFD_State := VFD_RUN_FORWARD;
	eStatusExp : E_VFD_Status := VFD_STATUS_READY_TO_RUN;
	bActiveExp : BOOL := TRUE;
	bBusyExp	: BOOL := TRUE;

END_VAR
TEST( 'When VFD_IDLE And IsStop Call Mr_RunForward Expect VFD_RUN_FORWARD');
IF nCycle >= nThCycle  THEN
	arrDataRead[0] := 20;
	FbVFDModbus.Convert( iRegionNo := 0,
						 pReadData := arrDataRead[0]);
	IF (FbVFDModbus.State = eStateFixture AND FbVFDModbus.isStop) OR FbVFDModbus.State = eStateExp  THEN
		FbVFDModbus.MR_RunForward( hz := 10	);				
		eStateACT := FbVFDModbus.State;
		//IF nCycle = (nThCycle + nCycleDuration-1) THEN
		AssertEquals( 	Expected := eStateExp,
							Actual := eStateACT,
							Message := 'TEST MR_RunForward failed at Change to VFD_RUN_FORWARD');
		bActiveACT := FbVFDModbus.Active;
		AssertEquals( Expected := bActiveExp,
						Actual := bActiveACT,
						Message := 'Test MR_RunForward Fail at Active');
		bBusyACT := FbVFDModbus.Busy;
		AssertEquals( Expected := bBusyExp,
						Actual := bBusyACT,
						Message := 'Test MR_RunForward Fail at Busy');
			TEST_FINISHED();	
		//END_IF

		
	ELSE
		eStateACT := FbVFDModbus.State;
		AssertEquals( 	Expected := eStateFixture,
						Actual := eStateACT,
						Message := 'FIXTURE CONDITION NOT PROPERLY AT STATE');
		bIsStopACT := FbVFDModbus.isStop;
		AssertEquals( 	Expected := bIsStopFixture,
						Actual := bIsStopACT,
						Message := 'FIXTURE CONDITION NOT PROPERLY AT properly IsStop');
		TEST_FINISHED();
	END_IF
END_IF
END_METHOD

METHOD PROTECTED WhenInitializingAndStatusReadyToRunExpectStateReadyInitialized
VAR_INPUT
	nThCycle : ULINT;// the cycle call implement
	nCycleDuration : UINT := 1;// number cycle this method be called
END_VAR
VAR
	bActiveACT : BOOL;
	bBusyACT	: BOOL;
	eStateACT : E_VFD_State;
	eStatusACT	: E_VFD_Status;
	//@TEST-FIXTURE
	eStateFixture	: E_VFD_State := VFD_INITIALIZING;
	//@TEST-EXPECT
	eStateExp	: E_VFD_State := VFD_READY_INITIALIZED;
	eStatusExp : E_VFD_Status := VFD_STATUS_READY_TO_RUN;
	bActiveExp : BOOL := FALSE;
	bBusyExp	: BOOL := TRUE;
END_VAR
TEST( 'When Initializing And Status is VFD_STATUS_READY_TO_RUN Expect State ReadyInitialized');
IF nCycle >= nThCycle THEN
	IF FbVFDModbus.State = eStateFixture OR FbVFDModbus.State = eStateExp THEN
		// Modbus Return Code and FBVFD must convert to Status Ready to Run
		arrDataRead[0] := 10;// suppose this value is will be converted to VFD_STATUS_READY_TO_RUN
		FbVFDModbus.Convert( iRegionNo := 0,
							pReadData := ADR( arrDataRead) );
		bActiveACT := FbVFDModbus.Active;
		AssertEquals( Expected := bActiveExp,
					Actual := bActiveACT,
					Message := 'Test MR_Init Fail at Active');
		bBusyACT := FbVFDModbus.Busy;
		AssertEquals( Expected := bBusyExp,
					Actual := bBusyACT,
					Message := ' Mr_Init Fail at Busy ');
		eStatusACT := FbVFDModbus.Status;
		AssertEquals( 	Expected := eStatusExp,
							Actual := eStatusACT,
							Message := 'TEST MR_Init failed at Convert to VFD_STATUS_READY_TO_RUN ');	
				
		IF nCycle = (nThCycle + nCycleDuration-1) THEN
			eStateACT := FbVFDModbus.State;
			AssertEquals( 	Expected := eStateExp,
							Actual := eStateACT,
							Message := 'TEST MR_Init failed at Change to VFD_READY_INITIALIZED ');
	
			TEST_FINISHED();	
		END_IF

		
	ELSE
		eStateACT := FbVFDModbus.State;
		AssertEquals( 	Expected := eStateFixture,
						Actual := eStateACT,
						Message := 'FIXTURE CONDITION NOT PROPERLY');
		TEST_FINISHED();
	END_IF
END_IF
END_METHOD

METHOD PROTECTED WhenInitializingExpectActiveFalseAndBusyTrue
VAR
	bActiveACT : BOOL;
	bBusyACT	: BOOL;
	eStateACT : E_VFD_State;
	//@TEST-FIXTURE
	eStateFixture	: E_VFD_State := VFD_INITIALIZING;
	//@TEST-EXPECT
	bActiveExp : BOOL := FALSE;
	bBusyExp	: BOOL := TRUE;
END_VAR
TEST( 'When Initializing expect Active is False and Busy is True');
IF FbVFDModbus.State = eStateFixture THEN
	// @TEST-RUN
	bBusyACT := FbVFDModbus.Busy;
	bActiveACT := FbVFDModbus.Active;
	// @TEST-ASSERT
	AssertEquals( Expected := bActiveExp,
					Actual := bActiveACT,
					Message := 'Test MR_Init Fail at Busy');
	AssertEquals( Expected := bBusyExp,
					Actual := bBusyACT,
					Message := ' Mr_Init Fail at Busy at Active');
	TEST_FINISHED();
ELSE
	eStateACT := FbVFDModbus.State;
	AssertEquals( Expected := eStateFixture,
					Actual := eStateACT,
					Message := 'FIXTURE CONDITION NOT PROPERLY');
	TEST_FINISHED();
END_IF
END_METHOD

METHOD PROTECTED WhenModbusNotRespondExpectVFD_STATUS_NOT_RESPOND

VAR
	eStatusACT	: E_VFD_Status;
	//@TEST-FIXTURE
		//MODBUS_ERRORS.MODBUSERROR_NO_RESPONSE;
	//@TEST-EXPECT
	eStatusExp : E_VFD_Status := VFD_STATUS_READY_TO_RUN;
END_VAR

FbVFDModbus.ModbusErrorID := MODBUS_ERRORS.MODBUSERROR_NO_RESPONSE;
END_METHOD

METHOD PROTECTED WhenModbusReturnFaultExpectVFD_STATUS_FAULT
VAR_INPUT
END_VAR
END_METHOD

METHOD PROTECTED WhenModbusReturnReadyToRunExpect_VFD_STATUS_READY_TO_RUN : BOOL
VAR_INPUT
END_VAR
END_METHOD

METHOD PROTECTED WhenModbusReturnRunningForwardExpectVFD_STATUS_RUNNING_FORWARD
VAR_INPUT
END_VAR
END_METHOD

METHOD PROTECTED WhenModbusReturnRunReverseExpectVFD_STATUS_RUNNING_REVERSE : BOOL
VAR_INPUT
END_VAR
END_METHOD

METHOD PROTECTED WhenModbusReturnStopExpectVFD_STATUS_STOP
VAR_INPUT
END_VAR
END_METHOD

METHOD PROTECTED WhenStateAlreadyInitializedAndCallMR_initExpectStateIsVFD_IDLE
VAR_INPUT
	nThCycle : ULINT;
	nCycleDuration :UINT;
END_VAR
VAR	
	bActiveACT : BOOL;
	bBusyACT	: BOOL;
	eStateACT : E_VFD_State;
	//@TEST-FIXTURE
	eStateFixture	: E_VFD_State := VFD_READY_INITIALIZED;
	//@TEST-EXPECT
	eStateExp	: E_VFD_State := VFD_IDLE;
	bActiveExp : BOOL := TRUE;
	bBusyExp	: BOOL := FALSE;
END_VAR
TEST( 'When VFD_READY_INITIALIZED and continuous call MR_Init Expect State VFD_IDLE and Busy is False and Active is True');
IF nCycle >= nThCycle THEN
	IF FbVFDModbus.State = eStateFixture OR FbVFDModbus.State = eStateExp THEN
		FbVFDModbus.MR_Init();
		eStateACT := FbVFDModbus.State;
		bActiveACT := FbVFDModbus.Active;
		bBusyACT := FbVFDModbus.Busy;
		AssertEquals( Expected := bBusyExp,
						Actual := bBusyACT,
						Message := 'TEST MR_Init at property Busy');
		IF nCycle = (nThCycle + nCycleDuration-1) THEN	
			AssertEquals( Expected := eStateExp,
							Actual := eStateACT,
							Message := 'TEST MR_Init at Goto VFD_IDLE');	
			AssertEquals( Expected := bActiveExp,
						Actual := bActiveACT,
						Message := 'TEST MR_Init at property Active');	
			TEST_FINISHED();	
		END_IF
	ELSE
		eStateACT := FbVFDModbus.State;
		AssertEquals( Expected := eStateFixture,
						Actual := eStateACT,
						Message := 'FIXTURE CONDITION NOT PROPERLY');
		TEST_FINISHED();
	END_IF
END_IF
END_METHOD

METHOD PROTECTED WhenUnInitializedExpect_Active_Busy_areFalse
VAR
	bActiveResult : BOOL;
	bBusyResult	: BOOL;
	eStateResult : E_VFD_State;
	//@TEST-FIXTURE
	eStateFixture	: E_VFD_State := VFD_UNINITIALIZED;
	//@TEST-EXPECT
	bActiveExp : BOOL := FALSE;
	bBusyExp	: BOOL := FALSE;
END_VAR
TEST( 'When UnInitialized expect Active and Busy are False');
IF FbVFDModbus.State = eStateFixture THEN
	// @TEST-RUN
	bBusyResult := FbVFDModbus.Busy;
	bActiveResult := FbVFDModbus.Active;
	// @TEST-ASSERT
	AssertEquals( Expected := bActiveExp,
					Actual := bActiveResult,
					Message := 'Test Uninitialized failed at Active');
	AssertEquals( Expected := bBusyExp,
					Actual := bBusyResult,
					Message := 'Test Uninitialized failed at Busy');
	TEST_FINISHED();
ELSE
	eStateResult := FbVFDModbus.State;
	AssertEquals( Expected := eStateFixture,
					Actual := eStateResult,
					Message := 'FIXTURE CONDITION NOT PROPERLY');
	TEST_FINISHED();
END_IF
END_METHOD

METHOD PROTECTED WhenUnInitializedMR_InitExpectStateInitializing
VAR
	eStateResult	: E_VFD_State;
	bBusyResult			: BOOL;
	//@TEST-FIXTURE
	eStateFixture	: E_VFD_State := VFD_UNINITIALIZED;
	//@TEST-EXPECT
	eStateExpect	: E_VFD_State := VFD_INITIALIZING;
	bBusyExpect	: BOOL := TRUE;
END_VAR
TEST( 'When UnInitialized call MR_Init Expect State Initializing and Busy is True');
IF FbVFDModbus.State = eStateFixture THEN
	// @TEST-RUN
	FbVFDModbus.MR_Init();
	eStateResult := FbVFDModbus.State;
	bBusyResult := FbVFDModbus.Busy;
	
	// @TEST-ASSERT
	AssertEquals( Expected := eStateExpect,
					Actual := eStateResult,
					Message := 'Test MR_Init Fail at Request');
	AssertEquals( Expected := bBusyExpect,
					Actual := bBusyResult,
					Message := 'Test Mr_Init Fail at Busy at Request');
	TEST_FINISHED();
ELSE
	eStateResult := FbVFDModbus.State;
	AssertEquals( Expected := eStateFixture,
					Actual := eStateResult,
					Message := 'FIXTURE CONDITION NOT PROPERLY');
	TEST_FINISHED();
END_IF
END_METHOD

METHOD PROTECTED WhenVFD_RUN_FORWARDAndVFD_STATUS_RUNFORWARDExpectVFD_RUNFORWARD_DONE
VAR_INPUT
	nThCycle : ULINT;// the cycle call implement
	nCycleDuration : UINT := 1;// number cycle this method be called
END_VAR
VAR
	bActiveACT : BOOL;
	bBusyACT	: BOOL;
	eStateACT : E_VFD_State;
	eStatusACT	: E_VFD_Status;
	//@TEST-FIXTURE
	eStateFixture	: E_VFD_State := VFD_RUN_FORWARD;
	//@TEST-EXPECT
	eStateExp	: E_VFD_State := VFD_RUN_FORWARD_DONE;
	eStatusExp : E_VFD_Status := VFD_STATUS_RUNNING_FORWARD;
	bActiveExp : BOOL := TRUE;
	bBusyExp	: BOOL := TRUE;
END_VAR
TEST( 'When VFD_RUN_FORWARD And VFD_STATUS_RUNFORWARD Expect VFD_RUNFORWARD_DONE');
IF nCycle >= nThCycle  THEN
	IF FbVFDModbus.State = eStateFixture  OR FbVFDModbus.State = eStateExp  THEN
		arrDataRead[0] := 20;// suppose this value is will be converted to VFD_STATUS_RUNNING_FORWARD
		FbVFDModbus.Convert( iRegionNo := 0,
							pReadData := ADR( arrDataRead) );
		eStatusACT := FbVFDModbus.Status;
		AssertEquals( 	Expected := eStatusExp,
							Actual := eStatusACT,
							Message := 'TEST  failed at Convert to VFD_RUN_FORWARD_DONE ');				
		eStateACT := FbVFDModbus.State;
		//IF nCycle = (nThCycle + nCycleDuration-1) THEN
		AssertEquals( 	Expected := eStateExp,
							Actual := eStateACT,
							Message := 'TEST MR_RunForward failed at Change to VFD_RUN_FORWARD_DONE');
		bActiveACT := FbVFDModbus.Active;
		AssertEquals( Expected := bActiveExp,
						Actual := bActiveACT,
						Message := 'Test MR_RunForward Fail at Active');
		bBusyACT := FbVFDModbus.Busy;
		AssertEquals( Expected := bBusyExp,
						Actual := bBusyACT,
						Message := 'Test MR_RunForward Fail at Busy');
			TEST_FINISHED();	
		//END_IF

		
	ELSE
		eStateACT := FbVFDModbus.State;
		AssertEquals( 	Expected := eStateFixture,
						Actual := eStateACT,
						Message := 'FIXTURE CONDITION NOT PROPERLY');
		TEST_FINISHED();
	END_IF
END_IF
END_METHOD

END_FUNCTION_BLOCK

// ---- TEST/PGR_Test.TcPOU
PROGRAM PGR_Test
VAR
	fbUniversalVfdModbusTest : FB_UniversalVFDModbus_Test;
END_VAR

TcUnit.RUN();

END_PROGRAM

// ---- TEST/README.TcPOU
FUNCTION README : bool

(*Chắc chắn rằng mỗi test case kiểm thử mức đơn vị sẽ độc lập với những test case khác.
 Không nên gọi một test case khác trong một test case. Test case không nên phụ thuộc vào nhau cả về data và thứ tự thực hiện.
Luôn luôn kiểm tra từng mô-đun một cách độc lập. 
Nếu không, sẽ có nhiều sự chồng chéo giữa các ca thử nghiệm và việc thay đổi đối với một đơn vị có thể ảnh hưởng đến tất cả các mô-đun
 khác và khiến phần mềm bị lỗi.
Đặt tên các đơn vị kiểm thử một cách rõ ràng và nhất quán. 
Đảm bảo rằng các test case dễ đọc, bất kỳ ai cũng có thể chọn test case và chạy nó mà không gặp bất kỳ vấn đề nào.
Khi triển khai việc thay đổi giao diện hoặc chức năng, 
cần chạy lại các test case trước đó nhằm đảm bảo việc thay đổi này không làm ảnh hưởng đến những test case cũ đã pass.
Luôn đảm bảo lỗi được xác định trong quá trình Unit test được sửa trước khi chuyển sang giai đoạn tiếp theo.
Không cố gắng viết test case để kiểm thử tất cả mọi thứ, thay vào đó nên tập chung vào kiểm thử sự ảnh hưởng của hành vi hệ thống
Bên cạnh viết test case để test hành vi hệ thống, cần viết thêm test case để kiểm thử hiệu năng của mã nguồn
Các testsuit nên đặt riêng ra, độc lập code với module
Không nên có nhiều assert trong một test case vì khi một điều kiện không thỏa mãn thì các assert khác sẽ bị bỏ qua
Sau một thời gian dài, số lượng test case nhiều, thời gian chạy lớn.
 Nên chia ra nhóm test case cũ và test case mới, test case cũ sẽ chạy với tần xuất ít hơn*)
 
(*Perspective:
So let's take a step back and ask what TDD is trying to help us with.
 TDD is trying to help us determine if our code is correct or not. And by correct,
 I mean "does the code meet the business requirements?" The selling point is that we know changes will be required in the future, 
and we want to make sure that our code remains correct after we make those changes.

I bring that perspective up because I think it's easy to get lost in the details and lose sight of what we're trying to achieve.

Principles - SAP:
While I'm not an expert in TDD, I think you're missing part of what Single Assertion Principle (SAP) is trying to teach.
 SAP can be restated as "test one thing at a time." But TOTAT doesn't roll off the tongue as easily as SAP does.

Testing one thing at a time means that you focus on one case; one path; one boundary condition; 
one error case; one whatever per test. 
And the driving idea behind that is you need to know what broke when the test case fails, so you can resolve the issue more quickly. 
If you test multiple conditions (ie. more than one thing) within a test and the test fails,
 then you have a lot more work on your hands. 
You first have to identify which of the multiple cases failed and then figure out why that case failed.
If you test one thing at a time, your search scope is a lot smaller and the defect is identified more quickly.
 Keep in mind that "test one thing at a time" doesn't necessarily exclude you from looking at more than one
 process output at a time. For example, when testing a "known good path", I may expect to see a specific,
 resulting value in foo as well as another value in bar and I may verify that foo != bar as part of my test. 
The key is to logically group the output checks based upon the case being tested.
Principles - PMP:
Likewise, I think you're missing a bit about what Private Method Principle (PMP) has to teach us. 
PMP encourages us to treat the system like a black box. For a given input, you should get a given output. 
You don't care how the black box generates the output. You only care that your outputs align with your inputs.

PMP is really good perspective for looking at the API aspects of your code. 
It can also help you scope what you have to test. 
Identify your interface points and verify that they meet the terms of their contracts. 
You don't need to care about how the behind-the-interface (aka private) methods do their job. 
You just need to verify they did what they were supposed to do.*)

END_FUNCTION
